// ---- POUs/LVCP2/PRG_LVCP2_CompensationCalculate.TcPOU
PROGRAM PRG_LVCP2_CompensationCalculate
VAR
    fbCompensationCalc : FB_CompensationCalculator;
    bCalculate : BOOL := TRUE;              // Sürekli hesaplama için
    nActiveGroups : INT := 10;              // Toplam 10 grup
    
    // Outputs
    stHMIData : ST_CompensationHMI;
    asCapacitorTags : ARRAY[0..99] OF STRING(30);
    nActiveTags : INT;
    
    // Özet bilgiler
    rTotalPower : REAL;
    nTotalCapacitors : INT;
    nActiveGroupCount : INT;
END_VAR

// Grup sayısını güncelle
GVL_LVCP1.nConfiguredGroups := nActiveGroups;

// Hesaplama
fbCompensationCalc(
    bExecute 				:= bCalculate,
    bGroupActive 			:= GVL_LVCP2.abGroupActive,
    stGroupConfig 			:= GVL_LVCP2.astCompensationGroups,
    nActiveGroups 			:= GVL_LVCP2.nConfiguredGroups,
    stHMI 					=> stHMIData,
    asActiveCapacitorTags 	=> asCapacitorTags,
    nActiveCapacitorCount 	=> nActiveTags
);

// Özet bilgiler
rTotalPower 		:= stHMIData.stSummary.rTotalActivePower;
nTotalCapacitors 	:= stHMIData.stSummary.nTotalActiveCapacitors;
nActiveGroupCount 	:= stHMIData.stSummary.nActiveGroupCount;

END_PROGRAM

// ---- POUs/LVCP2/PRG_LVCP2_MainDisconnector.TcPOU
PROGRAM PRG_LVCP2_MainDisconnector
VAR
    // Function Block Instance
    fbDisconnector		: FB_DisconnectorControl;
	
	stDisconnectorIO	: ST_DisconnectorIO;
	
    
    // Başlangıç konfigürasyonu için flag
    bInitDone: BOOL := FALSE;	
END_VAR

IF NOT bInitDone THEN
	bInitDone := TRUE;
	RETURN;
END_IF

//*************************************************************************
// Ana Besleme Ayırıcısı
// +EP7-8CB1
//*************************************************************************
fbDisconnector(
    // Fiziksel Girişler
    bContactorOn_FB 	:= stDisconnectorIO.bContactorOn_FB,
    bContactorOff_FB 	:= stDisconnectorIO.bContactorOff_FB,
    bLimitOn 			:= stDisconnectorIO.bLimitOn,
    bLimitOff 			:= stDisconnectorIO.bLimitOff,
    bThermalFault 		:= stDisconnectorIO.bThermalFault,
    bEarthSwitchOn 		:= stDisconnectorIO.bEarthSwitchOn,
    bEarthSwitchOff 	:= stDisconnectorIO.bEarthSwitchOff,
    bPLCControl 		:= stDisconnectorIO.bPLCControl,
    
    // Güvenlik Girişleri
    bSafetyLoop 		:= GVL_Alarm.bSafetyLoop,
    bInterlock 			:= FALSE,
    
    // Sistem Girişleri
    bMasterReset 		:= GVL_Alarm.bMasterReset,
    
    // HMI Bağlantısı
    stHMI 				:= GVL_LVCP2.stMainDisconnectorHMI,
    
    // Fiziksel Çıkışlar
    bContactorOn_Out 	=> stDisconnectorIO.bContactorOn_Out,
    bContactorOff_Out 	=> stDisconnectorIO.bContactorOff_Out
);

METHOD M_Init : BOOL
VAR_INPUT
END_VAR

GVL_LVCP1.stMainDisconnectorHMI.stConfig.bEarthSwitchExists := TRUE;
GVL_LVCP1.stMainDisconnectorHMI.stConfig.bGrounded := TRUE;
GVL_LVCP1.stMainDisconnectorHMI.stConfig.bInterlockEnable := TRUE;
GVL_LVCP1.stMainDisconnectorHMI.stConfig.dwOperationLimit := 10000;
GVL_LVCP1.stMainDisconnectorHMI.stConfig.nPhaseCount := 3;
GVL_LVCP1.stMainDisconnectorHMI.stConfig.rRatedCurrent := 1600.0;
GVL_LVCP1.stMainDisconnectorHMI.stConfig.rRatedVoltage := 1000.0;
GVL_LVCP1.stMainDisconnectorHMI.stConfig.sProductCode := '';
GVL_LVCP1.stMainDisconnectorHMI.stConfig.sProjectCode := '+EP7-8CB1';
GVL_LVCP1.stMainDisconnectorHMI.stConfig.tContactorDelay := T#500MS;
GVL_LVCP1.stMainDisconnectorHMI.stConfig.tMotionTimeout := T#50S;
END_METHOD

END_PROGRAM

// ---- POUs/LVCP2/PRG_LVCP2_Colors.TcPOU
PROGRAM PRG_LVCP2_Colors
VAR
	arrLine : ARRAY[1..4] OF E_LineColors;
	arrCapacitorSchemaColor : ARRAY[1..10] OF ST_CapacitorSchemaColorWithContactor;

	i : INT;
	bInitDone : BOOL;
END_VAR

IF NOT bInitDone THEN
	ACT_ContactorConfigurations();
	bInitDone := TRUE;
END_IF

//line1
arrLine[1] := E_LineColors.Energised_Red;

//line2
arrLine[2] := arrLine[1];

//line3
arrLine[3] := arrLine[2];

//line4
arrLine[4] := arrLine[3];

//şemaları kendi içerisinde kontrol edicez
FOR i:=1 TO 10 DO
	arrCapacitorSchemaColor[i].GroundColor := E_LineColors.Grounded_Green;
	arrCapacitorSchemaColor[i].BottomLineColor2 := E_LineColors.Grounded_Green;

	//topline
	arrCapacitorSchemaColor[i].TopLineColor := arrLine[4];
	
	//bottomLine - şema üzerinde ayırıcının altındaki her iki line birbiri ile bağlantılı olduğu için tek yerden yönetiliyor
	IF arrCapacitorSchemaColor[i].ContactorPosition = E_ContactorPosition.ON THEN
		arrCapacitorSchemaColor[i].BottomLineColor := arrCapacitorSchemaColor[i].TopLineColor;
	ELSE
		arrCapacitorSchemaColor[i].BottomLineColor := E_LineColors.Default;
	END_IF
	
	//capacitor
	arrCapacitorSchemaColor[i].CapacitorColor := arrCapacitorSchemaColor[i].BottomLineColor;
	
END_FOR

ACTION ACT_ContactorConfigurations:
arrCapacitorSchemaColor[1].ContactorPosition := GVL_LVCP2.stGroup1_ContactorHMI.stStatus.ePosition;
arrCapacitorSchemaColor[2].ContactorPosition := GVL_LVCP2.stGroup2_ContactorHMI.stStatus.ePosition;
arrCapacitorSchemaColor[3].ContactorPosition := GVL_LVCP2.stGroup3_ContactorHMI.stStatus.ePosition;
arrCapacitorSchemaColor[4].ContactorPosition := GVL_LVCP2.stGroup4_ContactorHMI.stStatus.ePosition;
arrCapacitorSchemaColor[5].ContactorPosition := GVL_LVCP2.stGroup5_ContactorHMI.stStatus.ePosition;
arrCapacitorSchemaColor[6].ContactorPosition := GVL_LVCP2.stGroup6_ContactorHMI.stStatus.ePosition;
arrCapacitorSchemaColor[7].ContactorPosition := GVL_LVCP2.stGroup7_ContactorHMI.stStatus.ePosition;
arrCapacitorSchemaColor[8].ContactorPosition := GVL_LVCP2.stGroup8_ContactorHMI.stStatus.ePosition;
arrCapacitorSchemaColor[9].ContactorPosition := GVL_LVCP2.stGroup9_ContactorHMI.stStatus.ePosition;
arrCapacitorSchemaColor[10].ContactorPosition := GVL_LVCP2.stGroup10_ContactorHMI.stStatus.ePosition;
END_ACTION

END_PROGRAM

// ---- POUs/LVCP2/PRG_LVCP2_Group1.TcPOU
PROGRAM PRG_LVCP2_Group1
VAR
    // Function Block Instance
    fbContactor: FB_ContactorControl;

    // Contactor 1 IO Structure  
    stContactor_IO: ST_ContactorIO;
    
    // Başlangıç konfigürasyonu için flag
    bContactorInitDone: BOOL := FALSE;
    bCapacitorInitDone: BOOL := FALSE;	
END_VAR



	M_Contactor();
	
	M_Capacitor();

METHOD M_Capacitor : BOOL
VAR
    nGroupIndex : INT;
END_VAR
	nGroupIndex := 0;  // Grup 1 için index
	
	IF NOT bCapacitorInitDone THEN
	
		// Grup 1 değerlerini ata
		GVL_LVCP2.astCompensationGroups[nGroupIndex].rPower := 25.0;
		GVL_LVCP2.astCompensationGroups[nGroupIndex].rVoltage := 450.0;
		GVL_LVCP2.astCompensationGroups[nGroupIndex].nQuantity := 10;
		GVL_LVCP2.astCompensationGroups[nGroupIndex].sTagPrefix := '+EP7-16C1';
		GVL_LVCP2.astCompensationGroups[nGroupIndex].sProductCode := 'ENT.CXD-450-25';
		
		bCapacitorInitDone := TRUE;
	END_IF
	
	// Grup 1 aktif durumu
	GVL_LVCP2.abGroupActive[nGroupIndex] := stContactor_IO.bFeedback;
	
	M_Capacitor := TRUE;
END_METHOD

METHOD M_Contactor : BOOL
VAR_INPUT
END_VAR
IF NOT bContactorInitDone THEN
    // Konfigürasyon parametreleri
    GVL_LVCP2.stGroup1_ContactorHMI.stConfig.sProjectCode := '+EP7-17K1';
    GVL_LVCP2.stGroup1_ContactorHMI.stConfig.sProductCode := 'ABB-1SFL637001R7011';
    GVL_LVCP2.stGroup1_ContactorHMI.stConfig.rRatedCurrent := 630.0;
    GVL_LVCP2.stGroup1_ContactorHMI.stConfig.rRatedVoltage := 1000.0;
    GVL_LVCP2.stGroup1_ContactorHMI.stConfig.nPhaseCount := 3;
    GVL_LVCP2.stGroup1_ContactorHMI.stConfig.tFeedbackDelay := T#500MS;
    GVL_LVCP2.stGroup1_ContactorHMI.stConfig.tWeldedDelay := T#2S;
    GVL_LVCP2.stGroup1_ContactorHMI.stConfig.dwOperationLimit := 100000;
    GVL_LVCP2.stGroup1_ContactorHMI.stConfig.bFeedbackRequired := FALSE;
    // Başlangıç bakım sayacı
    GVL_LVCP2.stGroup1_ContactorHMI.stStatistics.dwRemainingOperations := GVL_LVCP2.stGroup1_ContactorHMI.stConfig.dwOperationLimit;
	
	bContactorInitDone := TRUE;
END_IF	
	
// Function Block Çağrısı
fbContactor(
    // Fiziksel Girişler
    bFeedback 		:= stContactor_IO.bFeedback,
    bPLCControl 	:= stContactor_IO.bPLCControl,
    
    // Güvenlik Girişleri
    bSafetyLoop 	:= GVL_Alarm.bSafetyLoop,
    bInterlock 		:= FALSE,
    
    // Sistem Girişleri
    bMasterReset 	:= GVL_Alarm.bMasterReset,
    
    // HMI Bağlantısı
    stHMI 			:= GVL_LVCP2.stGroup1_ContactorHMI,
    
    // Fiziksel Çıkış
    bOutput 		=> stContactor_IO.bOutput
);

// SQL Kayıt İşlemi
IF GVL_LVCP2.stGroup1_ContactorHMI.stStatistics.bNewOperationFlag THEN
    // SQL kayıt fonksiyonunu çağır
    GVL_LVCP2.stGroup1_ContactorHMI.stStatistics.bNewOperationFlag := FALSE;
END_IF
END_METHOD

END_PROGRAM

// ---- POUs/LVCP2/PRG_LVCP2_Group2.TcPOU
PROGRAM PRG_LVCP2_Group2
VAR
    // Function Block Instance
    fbContactor: FB_ContactorControl;

    // Contactor 1 IO Structure  
    stContactor_IO: ST_ContactorIO;
    
    // Başlangıç konfigürasyonu için flag
    bContactorInitDone: BOOL := FALSE;
    bCapacitorInitDone: BOOL := FALSE;	
END_VAR



	M_Contactor();
	
	M_Capacitor();

METHOD M_Capacitor : BOOL
VAR
    nGroupIndex : INT;
END_VAR

nGroupIndex := 1;  // Grup 2 için index

IF NOT bCapacitorInitDone THEN
    // Grup 2 değerlerini ata
    GVL_LVCP2.astCompensationGroups[nGroupIndex].rPower := 25.0;
    GVL_LVCP2.astCompensationGroups[nGroupIndex].rVoltage := 450.0;
    GVL_LVCP2.astCompensationGroups[nGroupIndex].nQuantity := 8;
    GVL_LVCP2.astCompensationGroups[nGroupIndex].sTagPrefix := '+EP7-19C1';
    GVL_LVCP2.astCompensationGroups[nGroupIndex].sProductCode := 'ENT.CXD-450-25';
    
    bCapacitorInitDone := TRUE;
END_IF

// Grup 2 aktif durumu
GVL_LVCP2.abGroupActive[nGroupIndex] := stContactor_IO.bFeedback;

M_Capacitor := TRUE;
END_METHOD

METHOD M_Contactor : BOOL
VAR_INPUT
END_VAR

IF NOT bContactorInitDone THEN
    // Konfigürasyon parametreleri
    GVL_LVCP2.stGroup2_ContactorHMI.stConfig.sProjectCode := '+EP7-20K1';
    GVL_LVCP2.stGroup2_ContactorHMI.stConfig.sProductCode := 'ABB-1SFL597001R7011';
    GVL_LVCP2.stGroup2_ContactorHMI.stConfig.rRatedCurrent := 500.0;
    GVL_LVCP2.stGroup2_ContactorHMI.stConfig.rRatedVoltage := 1000.0;
    GVL_LVCP2.stGroup2_ContactorHMI.stConfig.nPhaseCount := 3;
    GVL_LVCP2.stGroup2_ContactorHMI.stConfig.tFeedbackDelay := T#500MS;
    GVL_LVCP2.stGroup2_ContactorHMI.stConfig.tWeldedDelay := T#2S;
    GVL_LVCP2.stGroup2_ContactorHMI.stConfig.dwOperationLimit := 100000;
    
    // Başlangıç bakım sayacı
    GVL_LVCP2.stGroup2_ContactorHMI.stStatistics.dwRemainingOperations := GVL_LVCP2.stGroup2_ContactorHMI.stConfig.dwOperationLimit;
    
    bContactorInitDone := TRUE;
END_IF

// Function Block Çağrısı
fbContactor(
    // Fiziksel Girişler
    bFeedback := stContactor_IO.bFeedback,
    bPLCControl := stContactor_IO.bPLCControl,
    
    // Güvenlik Girişleri
    bSafetyLoop := GVL_Alarm.bSafetyLoop,
    bInterlock := FALSE,
    
    // Sistem Girişleri
    bMasterReset := GVL_Alarm.bMasterReset,
    
    // HMI Bağlantısı
    stHMI := GVL_LVCP2.stGroup2_ContactorHMI,
    
    // Fiziksel Çıkış
    bOutput => stContactor_IO.bOutput
);

M_Contactor := TRUE;
END_METHOD

END_PROGRAM

// ---- POUs/LVCP2/PRG_LVCP2_Group3.TcPOU
PROGRAM PRG_LVCP2_Group3
VAR
    // Function Block Instance
    fbContactor: FB_ContactorControl;

    // Contactor 1 IO Structure  
    stContactor_IO: ST_ContactorIO;
    
    // Başlangıç konfigürasyonu için flag
    bContactorInitDone: BOOL := FALSE;
    bCapacitorInitDone: BOOL := FALSE;	
END_VAR



	M_Contactor();
	
	M_Capacitor();

METHOD M_Capacitor : BOOL
VAR
    nGroupIndex : INT;
END_VAR

nGroupIndex := 2;  // Grup 3 için index

IF NOT bCapacitorInitDone THEN
    // Grup 3 değerlerini ata
    GVL_LVCP2.astCompensationGroups[nGroupIndex].rPower := 25.0;
    GVL_LVCP2.astCompensationGroups[nGroupIndex].rVoltage := 450.0;
    GVL_LVCP2.astCompensationGroups[nGroupIndex].nQuantity := 6;
    GVL_LVCP2.astCompensationGroups[nGroupIndex].sTagPrefix := '+EP7-22C1';
    GVL_LVCP2.astCompensationGroups[nGroupIndex].sProductCode := 'ENT.CXD-450-25';
    
    bCapacitorInitDone := TRUE;
END_IF

// Grup 3 aktif durumu
GVL_LVCP2.abGroupActive[nGroupIndex] := stContactor_IO.bFeedback;

M_Capacitor := TRUE;
END_METHOD

METHOD M_Contactor : BOOL
VAR_INPUT
END_VAR
IF NOT bContactorInitDone THEN
    // Konfigürasyon parametreleri
    GVL_LVCP2.stGroup3_ContactorHMI.stConfig.sProjectCode := '+EP7-23K1';
    GVL_LVCP2.stGroup3_ContactorHMI.stConfig.sProductCode := 'ABB-1SFL597001R7011';
    GVL_LVCP2.stGroup3_ContactorHMI.stConfig.rRatedCurrent := 500.0;
    GVL_LVCP2.stGroup3_ContactorHMI.stConfig.rRatedVoltage := 1000.0;
    GVL_LVCP2.stGroup3_ContactorHMI.stConfig.nPhaseCount := 3;
    GVL_LVCP2.stGroup3_ContactorHMI.stConfig.tFeedbackDelay := T#500MS;
    GVL_LVCP2.stGroup3_ContactorHMI.stConfig.tWeldedDelay := T#2S;
    GVL_LVCP2.stGroup3_ContactorHMI.stConfig.dwOperationLimit := 100000;
    
    // Başlangıç bakım sayacı
    GVL_LVCP2.stGroup3_ContactorHMI.stStatistics.dwRemainingOperations := GVL_LVCP2.stGroup3_ContactorHMI.stConfig.dwOperationLimit;
    
    bContactorInitDone := TRUE;
END_IF

// Function Block Çağrısı
fbContactor(
    // Fiziksel Girişler
    bFeedback := stContactor_IO.bFeedback,
    bPLCControl := stContactor_IO.bPLCControl,
    
    // Güvenlik Girişleri
    bSafetyLoop := GVL_Alarm.bSafetyLoop,
    bInterlock := FALSE,
    
    // Sistem Girişleri
    bMasterReset := GVL_Alarm.bMasterReset,
    
    // HMI Bağlantısı
    stHMI := GVL_LVCP2.stGroup3_ContactorHMI,
    
    // Fiziksel Çıkış
    bOutput => stContactor_IO.bOutput
);

M_Contactor := TRUE;
END_METHOD

END_PROGRAM

// ---- POUs/LVCP2/PRG_LVCP2_Group4.TcPOU
PROGRAM PRG_LVCP2_Group4
VAR
    // Function Block Instance
    fbContactor: FB_ContactorControl;

    // Contactor 1 IO Structure  
    stContactor_IO: ST_ContactorIO;
    
    // Başlangıç konfigürasyonu için flag
    bContactorInitDone: BOOL := FALSE;
    bCapacitorInitDone: BOOL := FALSE;	
END_VAR



	M_Contactor();
	
	M_Capacitor();

METHOD M_Capacitor : BOOL
VAR
    nGroupIndex : INT;
END_VAR

nGroupIndex := 3;  // Grup 4 için index

IF NOT bCapacitorInitDone THEN
    // Grup 4 değerlerini ata
    GVL_LVCP2.astCompensationGroups[nGroupIndex].rPower := 25.0;
    GVL_LVCP2.astCompensationGroups[nGroupIndex].rVoltage := 450.0;
    GVL_LVCP2.astCompensationGroups[nGroupIndex].nQuantity := 5;
    GVL_LVCP2.astCompensationGroups[nGroupIndex].sTagPrefix := '+EP7-25C1';
    GVL_LVCP2.astCompensationGroups[nGroupIndex].sProductCode := 'ENT.CXD-450-25';
    
    bCapacitorInitDone := TRUE;
END_IF

// Grup 4 aktif durumu
GVL_LVCP2.abGroupActive[nGroupIndex] := stContactor_IO.bFeedback;

M_Capacitor := TRUE;
END_METHOD

METHOD M_Contactor : BOOL
VAR_INPUT
END_VAR
IF NOT bContactorInitDone THEN
    // Konfigürasyon parametreleri
    GVL_LVCP2.stGroup4_ContactorHMI.stConfig.sProjectCode := '+EP7-26K1';
    GVL_LVCP2.stGroup4_ContactorHMI.stConfig.sProductCode := 'ABB-1SFL597001R7011';
    GVL_LVCP2.stGroup4_ContactorHMI.stConfig.rRatedCurrent := 500.0;
    GVL_LVCP2.stGroup4_ContactorHMI.stConfig.rRatedVoltage := 1000.0;
    GVL_LVCP2.stGroup4_ContactorHMI.stConfig.nPhaseCount := 3;
    GVL_LVCP2.stGroup4_ContactorHMI.stConfig.tFeedbackDelay := T#500MS;
    GVL_LVCP2.stGroup4_ContactorHMI.stConfig.tWeldedDelay := T#2S;
    GVL_LVCP2.stGroup4_ContactorHMI.stConfig.dwOperationLimit := 100000;
    
    // Başlangıç bakım sayacı
    GVL_LVCP2.stGroup4_ContactorHMI.stStatistics.dwRemainingOperations := GVL_LVCP2.stGroup4_ContactorHMI.stConfig.dwOperationLimit;
    
    bContactorInitDone := TRUE;
END_IF

// Function Block Çağrısı
fbContactor(
    // Fiziksel Girişler
    bFeedback := stContactor_IO.bFeedback,
    bPLCControl := stContactor_IO.bPLCControl,
    
    // Güvenlik Girişleri
    bSafetyLoop := GVL_Alarm.bSafetyLoop,
    bInterlock := FALSE,
    
    // Sistem Girişleri
    bMasterReset := GVL_Alarm.bMasterReset,
    
    // HMI Bağlantısı
    stHMI := GVL_LVCP2.stGroup4_ContactorHMI,
    
    // Fiziksel Çıkış
    bOutput => stContactor_IO.bOutput
);

M_Contactor := TRUE;
END_METHOD

END_PROGRAM

// ---- POUs/LVCP2/PRG_LVCP2_Group5.TcPOU
PROGRAM PRG_LVCP2_Group5
VAR
    // Function Block Instance
    fbContactor: FB_ContactorControl;

    // Contactor 1 IO Structure  
    stContactor_IO: ST_ContactorIO;
    
    // Başlangıç konfigürasyonu için flag
    bContactorInitDone: BOOL := FALSE;
    bCapacitorInitDone: BOOL := FALSE;	
END_VAR



	M_Contactor();
	
	M_Capacitor();

METHOD M_Capacitor : BOOL
VAR
    nGroupIndex : INT;
END_VAR

nGroupIndex := 4;  // Grup 5 için index

IF NOT bCapacitorInitDone THEN
    // Grup 5 değerlerini ata
    GVL_LVCP2.astCompensationGroups[nGroupIndex].rPower := 25.0;
    GVL_LVCP2.astCompensationGroups[nGroupIndex].rVoltage := 450.0;
    GVL_LVCP2.astCompensationGroups[nGroupIndex].nQuantity := 4;
    GVL_LVCP2.astCompensationGroups[nGroupIndex].sTagPrefix := '+EP7-28C1';
    GVL_LVCP2.astCompensationGroups[nGroupIndex].sProductCode := 'ENT.CXD-450-25';
    
    bCapacitorInitDone := TRUE;
END_IF

// Grup 5 aktif durumu
GVL_LVCP2.abGroupActive[nGroupIndex] := stContactor_IO.bFeedback;

M_Capacitor := TRUE;
END_METHOD

METHOD M_Contactor : BOOL
VAR_INPUT
END_VAR
IF NOT bContactorInitDone THEN
    // Konfigürasyon parametreleri
    GVL_LVCP2.stGroup5_ContactorHMI.stConfig.sProjectCode := '+EP7-29K1';
    GVL_LVCP2.stGroup5_ContactorHMI.stConfig.sProductCode := 'ABB 1SFL547002R1311';
    GVL_LVCP2.stGroup5_ContactorHMI.stConfig.rRatedCurrent := 265.0;
    GVL_LVCP2.stGroup5_ContactorHMI.stConfig.rRatedVoltage := 1000.0;
    GVL_LVCP2.stGroup5_ContactorHMI.stConfig.nPhaseCount := 3;
    GVL_LVCP2.stGroup5_ContactorHMI.stConfig.tFeedbackDelay := T#500MS;
    GVL_LVCP2.stGroup5_ContactorHMI.stConfig.tWeldedDelay := T#2S;
    GVL_LVCP2.stGroup5_ContactorHMI.stConfig.dwOperationLimit := 100000;
    
    // Başlangıç bakım sayacı
    GVL_LVCP2.stGroup5_ContactorHMI.stStatistics.dwRemainingOperations := GVL_LVCP2.stGroup5_ContactorHMI.stConfig.dwOperationLimit;
    
    bContactorInitDone := TRUE;
END_IF

// Function Block Çağrısı
fbContactor(
    // Fiziksel Girişler
    bFeedback := stContactor_IO.bFeedback,
    bPLCControl := stContactor_IO.bPLCControl,
    
    // Güvenlik Girişleri
    bSafetyLoop := GVL_Alarm.bSafetyLoop,
    bInterlock := FALSE,
    
    // Sistem Girişleri
    bMasterReset := GVL_Alarm.bMasterReset,
    
    // HMI Bağlantısı
    stHMI := GVL_LVCP2.stGroup5_ContactorHMI,
    
    // Fiziksel Çıkış
    bOutput => stContactor_IO.bOutput
);

M_Contactor := TRUE;
END_METHOD

END_PROGRAM

// ---- POUs/LVCP2/PRG_LVCP2_Group6.TcPOU
PROGRAM PRG_LVCP2_Group6
VAR
    // Function Block Instance
    fbContactor: FB_ContactorControl;

    // Contactor 1 IO Structure  
    stContactor_IO: ST_ContactorIO;
    
    // Başlangıç konfigürasyonu için flag
    bContactorInitDone: BOOL := FALSE;
    bCapacitorInitDone: BOOL := FALSE;	
END_VAR



	M_Contactor();
	
	M_Capacitor();

METHOD M_Capacitor : BOOL
VAR
    nGroupIndex : INT;
END_VAR

nGroupIndex := 5;  // Grup 6 için index

IF NOT bCapacitorInitDone THEN
    // Grup 6 değerlerini ata
    GVL_LVCP2.astCompensationGroups[nGroupIndex].rPower := 25.0;
    GVL_LVCP2.astCompensationGroups[nGroupIndex].rVoltage := 450.0;
    GVL_LVCP2.astCompensationGroups[nGroupIndex].nQuantity := 3;
    GVL_LVCP2.astCompensationGroups[nGroupIndex].sTagPrefix := '+EP7-31C1';
    GVL_LVCP2.astCompensationGroups[nGroupIndex].sProductCode := 'ENT.CXD-450-25';
    
    bCapacitorInitDone := TRUE;
END_IF

// Grup 6 aktif durumu
GVL_LVCP2.abGroupActive[nGroupIndex] := stContactor_IO.bFeedback;

M_Capacitor := TRUE;
END_METHOD

METHOD M_Contactor : BOOL
VAR_INPUT
END_VAR
IF NOT bContactorInitDone THEN
    // Konfigürasyon parametreleri
    GVL_LVCP2.stGroup6_ContactorHMI.stConfig.sProjectCode := '+EP7-30K1';
    GVL_LVCP2.stGroup6_ContactorHMI.stConfig.sProductCode := 'ABB 1SFL547002R1311';
    GVL_LVCP2.stGroup6_ContactorHMI.stConfig.rRatedCurrent := 265.0;
    GVL_LVCP2.stGroup6_ContactorHMI.stConfig.rRatedVoltage := 1000.0;
    GVL_LVCP2.stGroup6_ContactorHMI.stConfig.nPhaseCount := 3;
    GVL_LVCP2.stGroup6_ContactorHMI.stConfig.tFeedbackDelay := T#500MS;
    GVL_LVCP2.stGroup6_ContactorHMI.stConfig.tWeldedDelay := T#2S;
    GVL_LVCP2.stGroup6_ContactorHMI.stConfig.dwOperationLimit := 100000;
    
    // Başlangıç bakım sayacı
    GVL_LVCP2.stGroup6_ContactorHMI.stStatistics.dwRemainingOperations := GVL_LVCP2.stGroup6_ContactorHMI.stConfig.dwOperationLimit;
    
    bContactorInitDone := TRUE;
END_IF

// Function Block Çağrısı
fbContactor(
    // Fiziksel Girişler
    bFeedback := stContactor_IO.bFeedback,
    bPLCControl := stContactor_IO.bPLCControl,
    
    // Güvenlik Girişleri
    bSafetyLoop := GVL_Alarm.bSafetyLoop,
    bInterlock := FALSE,
    
    // Sistem Girişleri
    bMasterReset := GVL_Alarm.bMasterReset,
    
    // HMI Bağlantısı
    stHMI := GVL_LVCP2.stGroup6_ContactorHMI,
    
    // Fiziksel Çıkış
    bOutput => stContactor_IO.bOutput
);

M_Contactor := TRUE;
END_METHOD

END_PROGRAM

// ---- POUs/LVCP2/PRG_LVCP2_Group7.TcPOU
PROGRAM PRG_LVCP2_Group7
VAR
    // Function Block Instance
    fbContactor: FB_ContactorControl;

    // Contactor 1 IO Structure  
    stContactor_IO: ST_ContactorIO;
    
    // Başlangıç konfigürasyonu için flag
    bContactorInitDone: BOOL := FALSE;
    bCapacitorInitDone: BOOL := FALSE;	
END_VAR



	M_Contactor();
	
	M_Capacitor();

METHOD M_Capacitor : BOOL
VAR
    nGroupIndex : INT;
END_VAR

nGroupIndex := 6;  // Grup 7 için index

IF NOT bCapacitorInitDone THEN
    // Grup 7 değerlerini ata
    GVL_LVCP2.astCompensationGroups[nGroupIndex].rPower := 25.0;
    GVL_LVCP2.astCompensationGroups[nGroupIndex].rVoltage := 450.0;
    GVL_LVCP2.astCompensationGroups[nGroupIndex].nQuantity := 2;
    GVL_LVCP2.astCompensationGroups[nGroupIndex].sTagPrefix := '+EP7-34C1';
    GVL_LVCP2.astCompensationGroups[nGroupIndex].sProductCode := 'ENT.CXD-450-25';
    
    bCapacitorInitDone := TRUE;
END_IF

// Grup 7 aktif durumu
GVL_LVCP2.abGroupActive[nGroupIndex] := stContactor_IO.bFeedback;

M_Capacitor := TRUE;
END_METHOD

METHOD M_Contactor : BOOL
VAR_INPUT
END_VAR
IF NOT bContactorInitDone THEN
    // Konfigürasyon parametreleri
    GVL_LVCP2.stGroup7_ContactorHMI.stConfig.sProjectCode := '+EP7-35K1';
    GVL_LVCP2.stGroup7_ContactorHMI.stConfig.sProductCode := 'ABB 1SFL447001R1311';
    GVL_LVCP2.stGroup7_ContactorHMI.stConfig.rRatedCurrent := 150.0;
    GVL_LVCP2.stGroup7_ContactorHMI.stConfig.rRatedVoltage := 1000.0;
    GVL_LVCP2.stGroup7_ContactorHMI.stConfig.nPhaseCount := 3;
    GVL_LVCP2.stGroup7_ContactorHMI.stConfig.tFeedbackDelay := T#500MS;
    GVL_LVCP2.stGroup7_ContactorHMI.stConfig.tWeldedDelay := T#2S;
    GVL_LVCP2.stGroup7_ContactorHMI.stConfig.dwOperationLimit := 100000;
    
    // Başlangıç bakım sayacı
    GVL_LVCP2.stGroup7_ContactorHMI.stStatistics.dwRemainingOperations := GVL_LVCP2.stGroup7_ContactorHMI.stConfig.dwOperationLimit;
    
    bContactorInitDone := TRUE;
END_IF

// Function Block Çağrısı
fbContactor(
    // Fiziksel Girişler
    bFeedback := stContactor_IO.bFeedback,
    bPLCControl := stContactor_IO.bPLCControl,
    
    // Güvenlik Girişleri
    bSafetyLoop := GVL_Alarm.bSafetyLoop,
    bInterlock := FALSE,
    
    // Sistem Girişleri
    bMasterReset := GVL_Alarm.bMasterReset,
    
    // HMI Bağlantısı
    stHMI := GVL_LVCP2.stGroup7_ContactorHMI,
    
    // Fiziksel Çıkış
    bOutput => stContactor_IO.bOutput
);

M_Contactor := TRUE;
END_METHOD

END_PROGRAM

// ---- POUs/LVCP2/PRG_LVCP2_Group8.TcPOU
PROGRAM PRG_LVCP2_Group8
VAR
    // Function Block Instance
    fbContactor: FB_ContactorControl;

    // Contactor 1 IO Structure  
    stContactor_IO: ST_ContactorIO;
    
    // Başlangıç konfigürasyonu için flag
    bContactorInitDone: BOOL := FALSE;
    bCapacitorInitDone: BOOL := FALSE;	
END_VAR



	M_Contactor();
	
	M_Capacitor();

METHOD M_Capacitor : BOOL
VAR
    nGroupIndex : INT;
END_VAR

nGroupIndex := 7;  // Grup 8 için index

IF NOT bCapacitorInitDone THEN
    // Grup 8 değerlerini ata
    GVL_LVCP2.astCompensationGroups[nGroupIndex].rPower := 12.5;
    GVL_LVCP2.astCompensationGroups[nGroupIndex].rVoltage := 450.0;
    GVL_LVCP2.astCompensationGroups[nGroupIndex].nQuantity := 3;
    GVL_LVCP2.astCompensationGroups[nGroupIndex].sTagPrefix := '+EP7-37C1';
    GVL_LVCP2.astCompensationGroups[nGroupIndex].sProductCode := 'ENT.CXD-450-12.5';
    
    bCapacitorInitDone := TRUE;
END_IF

// Grup 8 aktif durumu
GVL_LVCP2.abGroupActive[nGroupIndex] := stContactor_IO.bFeedback;

M_Capacitor := TRUE;
END_METHOD

METHOD M_Contactor : BOOL
VAR_INPUT
END_VAR
IF NOT bContactorInitDone THEN
    // Konfigürasyon parametreleri
    GVL_LVCP2.stGroup8_ContactorHMI.stConfig.sProjectCode := '+EP7-38K1';
    GVL_LVCP2.stGroup8_ContactorHMI.stConfig.sProductCode := 'ABB 1SFL447001R1311';
    GVL_LVCP2.stGroup8_ContactorHMI.stConfig.rRatedCurrent := 115.0;
    GVL_LVCP2.stGroup8_ContactorHMI.stConfig.rRatedVoltage := 1000.0;
    GVL_LVCP2.stGroup8_ContactorHMI.stConfig.nPhaseCount := 3;
    GVL_LVCP2.stGroup8_ContactorHMI.stConfig.tFeedbackDelay := T#500MS;
    GVL_LVCP2.stGroup8_ContactorHMI.stConfig.tWeldedDelay := T#2S;
    GVL_LVCP2.stGroup8_ContactorHMI.stConfig.dwOperationLimit := 100000;
    
    // Başlangıç bakım sayacı
    GVL_LVCP2.stGroup8_ContactorHMI.stStatistics.dwRemainingOperations := GVL_LVCP2.stGroup8_ContactorHMI.stConfig.dwOperationLimit;
    
    bContactorInitDone := TRUE;
END_IF

// Function Block Çağrısı
fbContactor(
    // Fiziksel Girişler
    bFeedback := stContactor_IO.bFeedback,
    bPLCControl := stContactor_IO.bPLCControl,
    
    // Güvenlik Girişleri
    bSafetyLoop := GVL_Alarm.bSafetyLoop,
    bInterlock := FALSE,
    
    // Sistem Girişleri
    bMasterReset := GVL_Alarm.bMasterReset,
    
    // HMI Bağlantısı
    stHMI := GVL_LVCP2.stGroup8_ContactorHMI,
    
    // Fiziksel Çıkış
    bOutput => stContactor_IO.bOutput
);

M_Contactor := TRUE;
END_METHOD

END_PROGRAM

// ---- POUs/LVCP2/PRG_LVCP2_Group9.TcPOU
PROGRAM PRG_LVCP2_Group9
VAR
    // Function Block Instance
    fbContactor: FB_ContactorControl;

    // Contactor 1 IO Structure  
    stContactor_IO: ST_ContactorIO;
    
    // Başlangıç konfigürasyonu için flag
    bContactorInitDone: BOOL := FALSE;
    bCapacitorInitDone: BOOL := FALSE;	
END_VAR



	M_Contactor();
	
	M_Capacitor();

METHOD M_Capacitor : BOOL
VAR
    nGroupIndex : INT;
END_VAR

nGroupIndex := 8;  // Grup 9 için index

IF NOT bCapacitorInitDone THEN
    // Grup 9 değerlerini ata
    GVL_LVCP2.astCompensationGroups[nGroupIndex].rPower := 12.5;
    GVL_LVCP2.astCompensationGroups[nGroupIndex].rVoltage := 450.0;
    GVL_LVCP2.astCompensationGroups[nGroupIndex].nQuantity := 2;
    GVL_LVCP2.astCompensationGroups[nGroupIndex].sTagPrefix := '+EP7-40C1';
    GVL_LVCP2.astCompensationGroups[nGroupIndex].sProductCode := 'ENT.CXD-450-12.5';
    
    bCapacitorInitDone := TRUE;
END_IF

// Grup 9 aktif durumu
GVL_LVCP2.abGroupActive[nGroupIndex] := stContactor_IO.bFeedback;

M_Capacitor := TRUE;
END_METHOD

METHOD M_Contactor : BOOL
VAR_INPUT
END_VAR
IF NOT bContactorInitDone THEN
    // Konfigürasyon parametreleri
    GVL_LVCP2.stGroup9_ContactorHMI.stConfig.sProjectCode := '+EP7-41K1';
    GVL_LVCP2.stGroup9_ContactorHMI.stConfig.sProductCode := 'ABB 1SFL427001R1311';
    GVL_LVCP2.stGroup9_ContactorHMI.stConfig.rRatedCurrent := 115.0;
    GVL_LVCP2.stGroup9_ContactorHMI.stConfig.rRatedVoltage := 1000.0;
    GVL_LVCP2.stGroup9_ContactorHMI.stConfig.nPhaseCount := 3;
    GVL_LVCP2.stGroup9_ContactorHMI.stConfig.tFeedbackDelay := T#500MS;
    GVL_LVCP2.stGroup9_ContactorHMI.stConfig.tWeldedDelay := T#2S;
    GVL_LVCP2.stGroup9_ContactorHMI.stConfig.dwOperationLimit := 100000;
    
    // Başlangıç bakım sayacı
    GVL_LVCP2.stGroup9_ContactorHMI.stStatistics.dwRemainingOperations := GVL_LVCP2.stGroup9_ContactorHMI.stConfig.dwOperationLimit;
    
    bContactorInitDone := TRUE;
END_IF

// Function Block Çağrısı
fbContactor(
    // Fiziksel Girişler
    bFeedback := stContactor_IO.bFeedback,
    bPLCControl := stContactor_IO.bPLCControl,
    
    // Güvenlik Girişleri
    bSafetyLoop := GVL_Alarm.bSafetyLoop,
    bInterlock := FALSE,
    
    // Sistem Girişleri
    bMasterReset := GVL_Alarm.bMasterReset,
    
    // HMI Bağlantısı
    stHMI := GVL_LVCP2.stGroup9_ContactorHMI,
    
    // Fiziksel Çıkış
    bOutput => stContactor_IO.bOutput
);

M_Contactor := TRUE;
END_METHOD

END_PROGRAM

// ---- POUs/LVCP2/PRG_LVCP2_Group10.TcPOU
PROGRAM PRG_LVCP2_Group10
VAR
    // Function Block Instance
    fbContactor: FB_ContactorControl;

    // Contactor 1 IO Structure  
    stContactor_IO: ST_ContactorIO;
    
    // Başlangıç konfigürasyonu için flag
    bContactorInitDone: BOOL := FALSE;
    bCapacitorInitDone: BOOL := FALSE;	
END_VAR



	M_Contactor();
	
	M_Capacitor();

METHOD M_Capacitor : BOOL
VAR
    nGroupIndex : INT;
END_VAR

nGroupIndex := 9;  // Grup 10 için index

IF NOT bCapacitorInitDone THEN
    // Grup 10 değerlerini ata
    GVL_LVCP2.astCompensationGroups[nGroupIndex].rPower := 12.5;
    GVL_LVCP2.astCompensationGroups[nGroupIndex].rVoltage := 450.0;
    GVL_LVCP2.astCompensationGroups[nGroupIndex].nQuantity := 1;
    GVL_LVCP2.astCompensationGroups[nGroupIndex].sTagPrefix := '+EP7-43C1';
    GVL_LVCP2.astCompensationGroups[nGroupIndex].sProductCode := 'ENT.CXD-450-12.5';
    
    bCapacitorInitDone := TRUE;
END_IF

// Grup 10 aktif durumu
GVL_LVCP2.abGroupActive[nGroupIndex] := stContactor_IO.bFeedback;

M_Capacitor := TRUE;
END_METHOD

METHOD M_Contactor : BOOL
VAR_INPUT
END_VAR
IF NOT bContactorInitDone THEN
    // Konfigürasyon parametreleri
    GVL_LVCP2.stGroup10_ContactorHMI.stConfig.sProjectCode := '+EP7-43K1';
    GVL_LVCP2.stGroup10_ContactorHMI.stConfig.sProductCode := 'ABB 1SFL427001R1311';
    GVL_LVCP2.stGroup10_ContactorHMI.stConfig.rRatedCurrent := 115.0;
    GVL_LVCP2.stGroup10_ContactorHMI.stConfig.rRatedVoltage := 1000.0;
    GVL_LVCP2.stGroup10_ContactorHMI.stConfig.nPhaseCount := 3;
    GVL_LVCP2.stGroup10_ContactorHMI.stConfig.tFeedbackDelay := T#500MS;
    GVL_LVCP2.stGroup10_ContactorHMI.stConfig.tWeldedDelay := T#2S;
    GVL_LVCP2.stGroup10_ContactorHMI.stConfig.dwOperationLimit := 100000;
    
    // Başlangıç bakım sayacı
    GVL_LVCP2.stGroup10_ContactorHMI.stStatistics.dwRemainingOperations := GVL_LVCP2.stGroup10_ContactorHMI.stConfig.dwOperationLimit;
    
    bContactorInitDone := TRUE;
END_IF

// Function Block Çağrısı
fbContactor(
    // Fiziksel Girişler
    bFeedback := stContactor_IO.bFeedback,
    bPLCControl := stContactor_IO.bPLCControl,
    
    // Güvenlik Girişleri
    bSafetyLoop := GVL_Alarm.bSafetyLoop,
    bInterlock := FALSE,
    
    // Sistem Girişleri
    bMasterReset := GVL_Alarm.bMasterReset,
    
    // HMI Bağlantısı
    stHMI := GVL_LVCP2.stGroup10_ContactorHMI,
    
    // Fiziksel Çıkış
    bOutput => stContactor_IO.bOutput
);

M_Contactor := TRUE;
END_METHOD

END_PROGRAM

// ---- POUs/LVCP5/PRG_LVCP5.TcPOU
PROGRAM PRG_LVCP5
VAR
END_VAR

	PRG_LVCP5_PowerMeasurement();

 	PRG_LVCP5_CompensationCalculate();

	PRG_LVCP5_MainCircuitBreaker();
	
	PRG_LVCP5_Colors();
	
	PRG_LVCP5_Group1();
	
	PRG_LVCP5_Group2();
	
	PRG_LVCP5_Group3();	
	
	PRG_LVCP5_Group4();	

	PRG_LVCP5_Group5();	

	PRG_LVCP5_Group6();	

	PRG_LVCP5_Group7();

END_PROGRAM

// ---- POUs/LVCP5/PRG_LVCP5_PowerMeasurement.TcPOU
PROGRAM PRG_LVCP5_PowerMeasurement
VAR
	// Enerji Yönetimi
	fbEL3453	: FB_EL3453;	
	stEL3453	: stEL3453;
END_VAR


	fbEL3453(pOut := ADR(stEL3453));

END_PROGRAM

// ---- POUs/LVCP5/PRG_LVCP5_CompensationCalculate.TcPOU
PROGRAM PRG_LVCP5_CompensationCalculate
VAR
    fbCompensationCalc : FB_CompensationCalculator;
    bCalculate : BOOL := TRUE;              // Sürekli hesaplama için
    nActiveGroups : INT := 10;              // Toplam 10 grup
    
    // Outputs
    stHMIData : ST_CompensationHMI;
    asCapacitorTags : ARRAY[0..99] OF STRING(30);
    nActiveTags : INT;
    
    // Özet bilgiler
    rTotalPower : REAL;
    nTotalCapacitors : INT;
    nActiveGroupCount : INT;
END_VAR

// Grup sayısını güncelle
GVL_LVCP5.nConfiguredGroups := nActiveGroups;

// Hesaplama
fbCompensationCalc(
    bExecute 				:= bCalculate,
    bGroupActive 			:= GVL_LVCP5.abGroupActive,
    stGroupConfig 			:= GVL_LVCP5.astCompensationGroups,
    nActiveGroups 			:= GVL_LVCP5.nConfiguredGroups,
    stHMI 					=> stHMIData,
    asActiveCapacitorTags 	=> asCapacitorTags,
    nActiveCapacitorCount 	=> nActiveTags
);

// Özet bilgiler
rTotalPower 		:= stHMIData.stSummary.rTotalActivePower;
nTotalCapacitors 	:= stHMIData.stSummary.nTotalActiveCapacitors;
nActiveGroupCount 	:= stHMIData.stSummary.nActiveGroupCount;

END_PROGRAM

// ---- POUs/LVCP5/PRG_LVCP5_MainCircuitBreaker.TcPOU
PROGRAM PRG_LVCP5_MainCircuitBreaker
VAR
    // Function Block Instance
    fbCircuitBreaker	: FB_CircuitBreaker;
	
    // IO Structure
    stCircuitBreakerIO	: ST_CircuitBreakerIO;	
    
    // Başlangıç konfigürasyonu için flag
    bInitDone			: BOOL := FALSE;
END_VAR

IF NOT bInitDone THEN
	M_Init();
	bInitDone := TRUE;
END_IF

// Function Block Çağrısı
fbCircuitBreaker(
    // Fiziksel Girişler
    bPositionOn 		:= stCircuitBreakerIO.bPositionOn,
    bPositionOff 		:= stCircuitBreakerIO.bPositionOff,
    bPositionTripped 	:= stCircuitBreakerIO.bPositionTripped,
    bSpringCharged 		:= stCircuitBreakerIO.bSpringCharged,
    bPLCControl 		:= stCircuitBreakerIO.bPLCControl,
    
    // Güvenlik Girişleri
    bSafetyLoop 		:= GVL_Alarm.bSafetyLoop,
    bInterlock 			:= FALSE,
    
    // Sistem Girişleri
    bMasterReset 		:= GVL_Alarm.bMasterReset,
    
    // HMI Bağlantısı
    stHMI 				:= GVL_LVCP5.stMainCircuitBreakerHMI,
    
    // Fiziksel Çıkışlar
    bOnCommand 			=> stCircuitBreakerIO.bOnCommand,
    bOffCommand 		=> stCircuitBreakerIO.bOffCommand
);

// SQL Kayıt İşlemi
IF GVL_LVCP5.stMainCircuitBreakerHMI.stStatistics.bNewOperationFlag THEN
    // SQL kayıt fonksiyonunu çağır
    GVL_LVCP5.stMainCircuitBreakerHMI.stStatistics.bNewOperationFlag := FALSE;
END_IF

METHOD M_Init : BOOL
VAR_INPUT
END_VAR
    // Konfigürasyon parametreleri
    GVL_LVCP5.stMainCircuitBreakerHMI.stConfig.sProjectCode := '+EP8-6F1';
    GVL_LVCP5.stMainCircuitBreakerHMI.stConfig.sProductCode := 'ETN C63N32D630';
    GVL_LVCP5.stMainCircuitBreakerHMI.stConfig.rRatedCurrent := 630.0;
    GVL_LVCP5.stMainCircuitBreakerHMI.stConfig.rRatedVoltage := 1000.0;
    GVL_LVCP5.stMainCircuitBreakerHMI.stConfig.nPhaseCount := 3;
    GVL_LVCP5.stMainCircuitBreakerHMI.stConfig.tMotionTimeout := T#5S;
    GVL_LVCP5.stMainCircuitBreakerHMI.stConfig.tSpringChargeTimeout := T#30S;
    GVL_LVCP5.stMainCircuitBreakerHMI.stConfig.bSpringChargeRequired := FALSE;
    GVL_LVCP5.stMainCircuitBreakerHMI.stConfig.dwOperationLimit := 10000;
    
    // Başlangıç bakım sayacı
    GVL_LVCP5.stMainCircuitBreakerHMI.stStatistics.dwRemainingOperations := GVL_LVCP5.stMainCircuitBreakerHMI.stConfig.dwOperationLimit;
END_METHOD

END_PROGRAM

// ---- POUs/LVCP5/PRG_LVCP5_Colors.TcPOU
PROGRAM PRG_LVCP5_Colors
VAR
	arrLine : ARRAY[1..4] OF E_LineColors;
	arrCapacitorSchemaColor : ARRAY[1..7] OF ST_CapacitorSchemaColorWithContactor;

	i : INT;
	bInitDone : BOOL;
END_VAR

IF NOT bInitDone THEN
	ACT_ContactorConfigurations();
	bInitDone := TRUE;
END_IF

//line1
arrLine[1] := E_LineColors.Energised_Red;

//line2
arrLine[2] := arrLine[1];

//line3
arrLine[3] := arrLine[2];

//line4
arrLine[4] := arrLine[3];

//şemaları kendi içerisinde kontrol edicez
FOR i:=1 TO 10 DO
	arrCapacitorSchemaColor[i].GroundColor := E_LineColors.Grounded_Green;
	arrCapacitorSchemaColor[i].BottomLineColor2 := E_LineColors.Grounded_Green;

	//topline
	arrCapacitorSchemaColor[i].TopLineColor := arrLine[4];
	
	//bottomLine - şema üzerinde ayırıcının altındaki her iki line birbiri ile bağlantılı olduğu için tek yerden yönetiliyor
	IF arrCapacitorSchemaColor[i].ContactorPosition = E_ContactorPosition.ON THEN
		arrCapacitorSchemaColor[i].BottomLineColor := arrCapacitorSchemaColor[i].TopLineColor;
	ELSE
		arrCapacitorSchemaColor[i].BottomLineColor := E_LineColors.Default;
	END_IF
	
	//capacitor
	arrCapacitorSchemaColor[i].CapacitorColor := arrCapacitorSchemaColor[i].BottomLineColor;
	
END_FOR

ACTION ACT_ContactorConfigurations:
arrCapacitorSchemaColor[1].ContactorPosition := GVL_LVCP5.stGroup1_ContactorHMI.stStatus.ePosition;
arrCapacitorSchemaColor[2].ContactorPosition := GVL_LVCP5.stGroup2_ContactorHMI.stStatus.ePosition;
arrCapacitorSchemaColor[3].ContactorPosition := GVL_LVCP5.stGroup3_ContactorHMI.stStatus.ePosition;
arrCapacitorSchemaColor[4].ContactorPosition := GVL_LVCP5.stGroup4_ContactorHMI.stStatus.ePosition;
arrCapacitorSchemaColor[5].ContactorPosition := GVL_LVCP5.stGroup5_ContactorHMI.stStatus.ePosition;
arrCapacitorSchemaColor[6].ContactorPosition := GVL_LVCP5.stGroup6_ContactorHMI.stStatus.ePosition;
arrCapacitorSchemaColor[7].ContactorPosition := GVL_LVCP5.stGroup7_ContactorHMI.stStatus.ePosition;
END_ACTION

END_PROGRAM

// ---- POUs/LVCP5/PRG_LVCP5_Group1.TcPOU
PROGRAM PRG_LVCP5_Group1
VAR
    // Function Block Instance
    fbContactor: FB_ContactorControl;

    // Contactor 1 IO Structure  
    stContactor_IO: ST_ContactorIO;
    
    // Başlangıç konfigürasyonu için flag
    bContactorInitDone: BOOL := FALSE;
    bCapacitorInitDone: BOOL := FALSE;	
END_VAR



	M_Contactor();
	
	M_Capacitor();

METHOD M_Capacitor : BOOL
VAR
    nGroupIndex : INT;
END_VAR
	nGroupIndex := 0;  // Grup 1 için index
	
	IF NOT bCapacitorInitDone THEN
	
		// Grup 1 değerlerini ata
		GVL_LVCP5.astCompensationGroups[nGroupIndex].rPower := 10.0;
		GVL_LVCP5.astCompensationGroups[nGroupIndex].rVoltage := 450.0;
		GVL_LVCP5.astCompensationGroups[nGroupIndex].nQuantity := 10;
		GVL_LVCP5.astCompensationGroups[nGroupIndex].sTagPrefix := '+EP8-16C1';
		GVL_LVCP5.astCompensationGroups[nGroupIndex].sProductCode := 'ENT.CXD-450-10';
		
		bCapacitorInitDone := TRUE;
	END_IF
	
	// Grup 1 aktif durumu
	GVL_LVCP5.abGroupActive[nGroupIndex] := stContactor_IO.bFeedback;
	
	M_Capacitor := TRUE;
END_METHOD

METHOD M_Contactor : BOOL
VAR_INPUT
END_VAR
IF NOT bContactorInitDone THEN
    // Konfigürasyon parametreleri
    GVL_LVCP5.stGroup1_ContactorHMI.stConfig.sProjectCode := '+EP8-17K1';
    GVL_LVCP5.stGroup1_ContactorHMI.stConfig.sProductCode := 'SCH LC1G225LSEA';
    GVL_LVCP5.stGroup1_ContactorHMI.stConfig.rRatedCurrent := 225.0;
    GVL_LVCP5.stGroup1_ContactorHMI.stConfig.rRatedVoltage := 1000.0;
    GVL_LVCP5.stGroup1_ContactorHMI.stConfig.nPhaseCount := 3;
    GVL_LVCP5.stGroup1_ContactorHMI.stConfig.tFeedbackDelay := T#500MS;
    GVL_LVCP5.stGroup1_ContactorHMI.stConfig.tWeldedDelay := T#2S;
    GVL_LVCP5.stGroup1_ContactorHMI.stConfig.dwOperationLimit := 100000;
    
    // Başlangıç bakım sayacı
    GVL_LVCP5.stGroup1_ContactorHMI.stStatistics.dwRemainingOperations := GVL_LVCP5.stGroup1_ContactorHMI.stConfig.dwOperationLimit;
	
	bContactorInitDone := TRUE;
END_IF	
	
// Function Block Çağrısı
fbContactor(
    // Fiziksel Girişler
    bFeedback 		:= stContactor_IO.bFeedback,
    bPLCControl 	:= stContactor_IO.bPLCControl,
    
    // Güvenlik Girişleri
    bSafetyLoop 	:= GVL_Alarm.bSafetyLoop,
    bInterlock 		:= FALSE,
    
    // Sistem Girişleri
    bMasterReset 	:= GVL_Alarm.bMasterReset,
    
    // HMI Bağlantısı
    stHMI 			:= GVL_LVCP5.stGroup1_ContactorHMI,
    
    // Fiziksel Çıkış
    bOutput 		=> stContactor_IO.bOutput
);

// SQL Kayıt İşlemi
IF GVL_LVCP5.stGroup1_ContactorHMI.stStatistics.bNewOperationFlag THEN
    // SQL kayıt fonksiyonunu çağır
    GVL_LVCP5.stGroup1_ContactorHMI.stStatistics.bNewOperationFlag := FALSE;
END_IF
END_METHOD

END_PROGRAM

// ---- POUs/LVCP5/PRG_LVCP5_Group2.TcPOU
PROGRAM PRG_LVCP5_Group2
VAR
    // Function Block Instance
    fbContactor: FB_ContactorControl;

    // Contactor 1 IO Structure  
    stContactor_IO: ST_ContactorIO;
    
    // Başlangıç konfigürasyonu için flag
    bContactorInitDone: BOOL := FALSE;
    bCapacitorInitDone: BOOL := FALSE;	
END_VAR



	M_Contactor();
	
	M_Capacitor();

METHOD M_Capacitor : BOOL
VAR
    nGroupIndex : INT;
END_VAR

nGroupIndex := 1;  // Grup 2 için index

IF NOT bCapacitorInitDone THEN
    // Grup 2 değerlerini ata
    GVL_LVCP5.astCompensationGroups[nGroupIndex].rPower := 10.0;
    GVL_LVCP5.astCompensationGroups[nGroupIndex].rVoltage := 450.0;
    GVL_LVCP5.astCompensationGroups[nGroupIndex].nQuantity := 9;
    GVL_LVCP5.astCompensationGroups[nGroupIndex].sTagPrefix := '+EP8-19C1';
    GVL_LVCP5.astCompensationGroups[nGroupIndex].sProductCode := 'ENT.CXD-450-10';
    
    bCapacitorInitDone := TRUE;
END_IF

// Grup 2 aktif durumu
GVL_LVCP5.abGroupActive[nGroupIndex] := stContactor_IO.bFeedback;

M_Capacitor := TRUE;
END_METHOD

METHOD M_Contactor : BOOL
VAR_INPUT
END_VAR

IF NOT bContactorInitDone THEN
    // Konfigürasyon parametreleri
    GVL_LVCP5.stGroup2_ContactorHMI.stConfig.sProjectCode := '+EP6-20K1';
    GVL_LVCP5.stGroup2_ContactorHMI.stConfig.sProductCode := 'SCH LC1G500LSEA';
    GVL_LVCP5.stGroup2_ContactorHMI.stConfig.rRatedCurrent := 500.0;
    GVL_LVCP5.stGroup2_ContactorHMI.stConfig.rRatedVoltage := 1000.0;
    GVL_LVCP5.stGroup2_ContactorHMI.stConfig.nPhaseCount := 3;
    GVL_LVCP5.stGroup2_ContactorHMI.stConfig.tFeedbackDelay := T#500MS;
    GVL_LVCP5.stGroup2_ContactorHMI.stConfig.tWeldedDelay := T#2S;
    GVL_LVCP5.stGroup2_ContactorHMI.stConfig.dwOperationLimit := 100000;
    
    // Başlangıç bakım sayacı
    GVL_LVCP5.stGroup2_ContactorHMI.stStatistics.dwRemainingOperations := GVL_LVCP5.stGroup2_ContactorHMI.stConfig.dwOperationLimit;
    
    bContactorInitDone := TRUE;
END_IF

// Function Block Çağrısı
fbContactor(
    // Fiziksel Girişler
    bFeedback 		:= stContactor_IO.bFeedback,
    bPLCControl 	:= stContactor_IO.bPLCControl,
    
    // Güvenlik Girişleri
    bSafetyLoop 	:= GVL_Alarm.bSafetyLoop,
    bInterlock 		:= FALSE,
    
    // Sistem Girişleri
    bMasterReset 	:= GVL_Alarm.bMasterReset,
    
    // HMI Bağlantısı
    stHMI 			:= GVL_LVCP5.stGroup2_ContactorHMI,
    
    // Fiziksel Çıkış
    bOutput 		=> stContactor_IO.bOutput
);

M_Contactor := TRUE;
END_METHOD

END_PROGRAM

// ---- POUs/LVCP5/PRG_LVCP5_Group3.TcPOU
PROGRAM PRG_LVCP5_Group3
VAR
    // Function Block Instance
    fbContactor: FB_ContactorControl;

    // Contactor 1 IO Structure  
    stContactor_IO: ST_ContactorIO;
    
    // Başlangıç konfigürasyonu için flag
    bContactorInitDone: BOOL := FALSE;
    bCapacitorInitDone: BOOL := FALSE;	
END_VAR



	M_Contactor();
	
	M_Capacitor();

METHOD M_Capacitor : BOOL
VAR
    nGroupIndex : INT;
END_VAR

nGroupIndex := 2;  // Grup 3 için index

IF NOT bCapacitorInitDone THEN
    // Grup 3 değerlerini ata
    GVL_LVCP5.astCompensationGroups[nGroupIndex].rPower := 10.0;
    GVL_LVCP5.astCompensationGroups[nGroupIndex].rVoltage := 450.0;
    GVL_LVCP5.astCompensationGroups[nGroupIndex].nQuantity := 8;
    GVL_LVCP5.astCompensationGroups[nGroupIndex].sTagPrefix := '+EP8-22C1';
    GVL_LVCP5.astCompensationGroups[nGroupIndex].sProductCode := 'ENT.CXD-450-10';
    
    bCapacitorInitDone := TRUE;
END_IF

// Grup 3 aktif durumu
GVL_LVCP5.abGroupActive[nGroupIndex] := stContactor_IO.bFeedback;

M_Capacitor := TRUE;
END_METHOD

METHOD M_Contactor : BOOL
VAR_INPUT
END_VAR
IF NOT bContactorInitDone THEN
    // Konfigürasyon parametreleri
    GVL_LVCP5.stGroup3_ContactorHMI.stConfig.sProjectCode := '+EP8-23K1';
    GVL_LVCP5.stGroup3_ContactorHMI.stConfig.sProductCode := 'SCH LC1G185LSEA';
    GVL_LVCP5.stGroup3_ContactorHMI.stConfig.rRatedCurrent := 185.0;
    GVL_LVCP5.stGroup3_ContactorHMI.stConfig.rRatedVoltage := 1000.0;
    GVL_LVCP5.stGroup3_ContactorHMI.stConfig.nPhaseCount := 3;
    GVL_LVCP5.stGroup3_ContactorHMI.stConfig.tFeedbackDelay := T#500MS;
    GVL_LVCP5.stGroup3_ContactorHMI.stConfig.tWeldedDelay := T#2S;
    GVL_LVCP5.stGroup3_ContactorHMI.stConfig.dwOperationLimit := 100000;
    
    // Başlangıç bakım sayacı
    GVL_LVCP5.stGroup3_ContactorHMI.stStatistics.dwRemainingOperations := GVL_LVCP5.stGroup3_ContactorHMI.stConfig.dwOperationLimit;
    
    bContactorInitDone := TRUE;
END_IF

// Function Block Çağrısı
fbContactor(
    // Fiziksel Girişler
    bFeedback 		:= stContactor_IO.bFeedback,
    bPLCControl 	:= stContactor_IO.bPLCControl,
    
    // Güvenlik Girişleri
    bSafetyLoop 	:= GVL_Alarm.bSafetyLoop,
    bInterlock 		:= FALSE,
    
    // Sistem Girişleri
    bMasterReset 	:= GVL_Alarm.bMasterReset,
    
    // HMI Bağlantısı
    stHMI 			:= GVL_LVCP5.stGroup3_ContactorHMI,
    
    // Fiziksel Çıkış
    bOutput 		=> stContactor_IO.bOutput
);

M_Contactor := TRUE;
END_METHOD

END_PROGRAM

// ---- POUs/LVCP5/PRG_LVCP5_Group4.TcPOU
PROGRAM PRG_LVCP5_Group4
VAR
    // Function Block Instance
    fbContactor: FB_ContactorControl;

    // Contactor 1 IO Structure  
    stContactor_IO: ST_ContactorIO;
    
    // Başlangıç konfigürasyonu için flag
    bContactorInitDone: BOOL := FALSE;
    bCapacitorInitDone: BOOL := FALSE;	
END_VAR



	M_Contactor();
	
	M_Capacitor();

METHOD M_Capacitor : BOOL
VAR
    nGroupIndex : INT;
END_VAR

nGroupIndex := 3;  // Grup 4 için index

IF NOT bCapacitorInitDone THEN
    // Grup 4 değerlerini ata
    GVL_LVCP5.astCompensationGroups[nGroupIndex].rPower := 10.0;
    GVL_LVCP5.astCompensationGroups[nGroupIndex].rVoltage := 450.0;
    GVL_LVCP5.astCompensationGroups[nGroupIndex].nQuantity := 7;
    GVL_LVCP5.astCompensationGroups[nGroupIndex].sTagPrefix := '+EP8-25C1';
    GVL_LVCP5.astCompensationGroups[nGroupIndex].sProductCode := 'ENT.CXD-450-10';
    
    bCapacitorInitDone := TRUE;
END_IF

// Grup 4 aktif durumu
GVL_LVCP5.abGroupActive[nGroupIndex] := stContactor_IO.bFeedback;

M_Capacitor := TRUE;
END_METHOD

METHOD M_Contactor : BOOL
VAR_INPUT
END_VAR
IF NOT bContactorInitDone THEN
    // Konfigürasyon parametreleri
    GVL_LVCP5.stGroup4_ContactorHMI.stConfig.sProjectCode := '+EP8-26K1';
    GVL_LVCP5.stGroup4_ContactorHMI.stConfig.sProductCode := 'SCH LC1G150LSEA';
    GVL_LVCP5.stGroup4_ContactorHMI.stConfig.rRatedCurrent := 150.0;
    GVL_LVCP5.stGroup4_ContactorHMI.stConfig.rRatedVoltage := 1000.0;
    GVL_LVCP5.stGroup4_ContactorHMI.stConfig.nPhaseCount := 3;
    GVL_LVCP5.stGroup4_ContactorHMI.stConfig.tFeedbackDelay := T#500MS;
    GVL_LVCP5.stGroup4_ContactorHMI.stConfig.tWeldedDelay := T#2S;
    GVL_LVCP5.stGroup4_ContactorHMI.stConfig.dwOperationLimit := 100000;
    
    // Başlangıç bakım sayacı
    GVL_LVCP5.stGroup4_ContactorHMI.stStatistics.dwRemainingOperations := GVL_LVCP5.stGroup4_ContactorHMI.stConfig.dwOperationLimit;
    
    bContactorInitDone := TRUE;
END_IF

// Function Block Çağrısı
fbContactor(
    // Fiziksel Girişler
    bFeedback 		:= stContactor_IO.bFeedback,
    bPLCControl 	:= stContactor_IO.bPLCControl,
    
    // Güvenlik Girişleri
    bSafetyLoop 	:= GVL_Alarm.bSafetyLoop,
    bInterlock 		:= FALSE,
    
    // Sistem Girişleri
    bMasterReset 	:= GVL_Alarm.bMasterReset,
    
    // HMI Bağlantısı
    stHMI 			:= GVL_LVCP5.stGroup4_ContactorHMI,
    
    // Fiziksel Çıkış
    bOutput 		=> stContactor_IO.bOutput
);

M_Contactor := TRUE;
END_METHOD

END_PROGRAM

// ---- POUs/LVCP5/PRG_LVCP5_Group5.TcPOU
PROGRAM PRG_LVCP5_Group5
VAR
    // Function Block Instance
    fbContactor: FB_ContactorControl;

    // Contactor 1 IO Structure  
    stContactor_IO: ST_ContactorIO;
    
    // Başlangıç konfigürasyonu için flag
    bContactorInitDone: BOOL := FALSE;
    bCapacitorInitDone: BOOL := FALSE;	
END_VAR

	M_Contactor();
	
	M_Capacitor();

METHOD M_Capacitor : BOOL
VAR
    nGroupIndex : INT;
END_VAR

nGroupIndex := 4;  // Grup 5 için index

IF NOT bCapacitorInitDone THEN
    // Grup 5 değerlerini ata
    GVL_LVCP5.astCompensationGroups[nGroupIndex].rPower := 10.0;
    GVL_LVCP5.astCompensationGroups[nGroupIndex].rVoltage := 450.0;
    GVL_LVCP5.astCompensationGroups[nGroupIndex].nQuantity := 3;
    GVL_LVCP5.astCompensationGroups[nGroupIndex].sTagPrefix := '+EP8-28C1';
    GVL_LVCP5.astCompensationGroups[nGroupIndex].sProductCode := 'ENT.CXD-450-10';
    
    bCapacitorInitDone := TRUE;
END_IF

// Grup 5 aktif durumu
GVL_LVCP5.abGroupActive[nGroupIndex] := stContactor_IO.bFeedback;

M_Capacitor := TRUE;
END_METHOD

METHOD M_Contactor : BOOL
VAR_INPUT
END_VAR
bContactorInitDone := bContactorInitDone;
IF NOT bContactorInitDone THEN
    // Konfigürasyon parametreleri
    GVL_LVCP5.stGroup5_ContactorHMI.stConfig.sProjectCode := '+EP8-29K1';
    GVL_LVCP5.stGroup5_ContactorHMI.stConfig.sProductCode := 'SCH LC1D40A3P7';
    GVL_LVCP5.stGroup5_ContactorHMI.stConfig.rRatedCurrent := 40.0;
    GVL_LVCP5.stGroup5_ContactorHMI.stConfig.rRatedVoltage := 690.0;
    GVL_LVCP5.stGroup5_ContactorHMI.stConfig.nPhaseCount := 3;
    GVL_LVCP5.stGroup5_ContactorHMI.stConfig.tFeedbackDelay := T#500MS;
    GVL_LVCP5.stGroup5_ContactorHMI.stConfig.tWeldedDelay := T#2S;
    GVL_LVCP5.stGroup5_ContactorHMI.stConfig.dwOperationLimit := 100000;
    
    // Başlangıç bakım sayacı
    GVL_LVCP5.stGroup5_ContactorHMI.stStatistics.dwRemainingOperations := GVL_LVCP5.stGroup5_ContactorHMI.stConfig.dwOperationLimit;
    
    bContactorInitDone := TRUE;
END_IF

// Function Block Çağrısı
fbContactor(
    // Fiziksel Girişler
    bFeedback 		:= stContactor_IO.bFeedback,
    bPLCControl 	:= stContactor_IO.bPLCControl,
    
    // Güvenlik Girişleri
    bSafetyLoop 	:= GVL_Alarm.bSafetyLoop,
    bInterlock 		:= FALSE,
    
    // Sistem Girişleri
    bMasterReset 	:= GVL_Alarm.bMasterReset,
    
    // HMI Bağlantısı
    stHMI 			:= GVL_LVCP5.stGroup5_ContactorHMI,
    
    // Fiziksel Çıkış
    bOutput 		=> stContactor_IO.bOutput
);

M_Contactor := TRUE;
END_METHOD

END_PROGRAM

// ---- POUs/LVCP5/PRG_LVCP5_Group6.TcPOU
PROGRAM PRG_LVCP5_Group6
VAR
    // Function Block Instance
    fbContactor: FB_ContactorControl;

    // Contactor 1 IO Structure  
    stContactor_IO: ST_ContactorIO;
    
    // Başlangıç konfigürasyonu için flag
    bContactorInitDone: BOOL := FALSE;
    bCapacitorInitDone: BOOL := FALSE;	
END_VAR



	M_Contactor();
	
	M_Capacitor();

METHOD M_Capacitor : BOOL
VAR
    nGroupIndex : INT;
END_VAR

nGroupIndex := 5;  // Grup 6 için index

IF NOT bCapacitorInitDone THEN
    // Grup 6 değerlerini ata
    GVL_LVCP5.astCompensationGroups[nGroupIndex].rPower := 25.0;
    GVL_LVCP5.astCompensationGroups[nGroupIndex].rVoltage := 450.0;
    GVL_LVCP5.astCompensationGroups[nGroupIndex].nQuantity := 2;
    GVL_LVCP5.astCompensationGroups[nGroupIndex].sTagPrefix := '+EP8-31C1';
    GVL_LVCP5.astCompensationGroups[nGroupIndex].sProductCode := 'ENT.CXD-450-10';
    
    bCapacitorInitDone := TRUE;
END_IF

// Grup 6 aktif durumu
GVL_LVCP5.abGroupActive[nGroupIndex] := stContactor_IO.bFeedback;

M_Capacitor := TRUE;
END_METHOD

METHOD M_Contactor : BOOL
VAR_INPUT
END_VAR
IF NOT bContactorInitDone THEN
    // Konfigürasyon parametreleri
    GVL_LVCP5.stGroup6_ContactorHMI.stConfig.sProjectCode := '+EP8-32K1';
    GVL_LVCP5.stGroup6_ContactorHMI.stConfig.sProductCode := 'SCH LC1D40A3P7';
    GVL_LVCP5.stGroup6_ContactorHMI.stConfig.rRatedCurrent := 40.0;
    GVL_LVCP5.stGroup6_ContactorHMI.stConfig.rRatedVoltage := 690.0;
    GVL_LVCP5.stGroup6_ContactorHMI.stConfig.nPhaseCount := 3;
    GVL_LVCP5.stGroup6_ContactorHMI.stConfig.tFeedbackDelay := T#500MS;
    GVL_LVCP5.stGroup6_ContactorHMI.stConfig.tWeldedDelay := T#2S;
    GVL_LVCP5.stGroup6_ContactorHMI.stConfig.dwOperationLimit := 100000;
    
    // Başlangıç bakım sayacı
    GVL_LVCP5.stGroup6_ContactorHMI.stStatistics.dwRemainingOperations := GVL_LVCP5.stGroup6_ContactorHMI.stConfig.dwOperationLimit;
    
    bContactorInitDone := TRUE;
END_IF

// Function Block Çağrısı
fbContactor(
    // Fiziksel Girişler
    bFeedback 		:= stContactor_IO.bFeedback,
    bPLCControl 	:= stContactor_IO.bPLCControl,
    
    // Güvenlik Girişleri
    bSafetyLoop 	:= GVL_Alarm.bSafetyLoop,
    bInterlock 		:= FALSE,
    
    // Sistem Girişleri
    bMasterReset 	:= GVL_Alarm.bMasterReset,
    
    // HMI Bağlantısı
    stHMI 			:= GVL_LVCP5.stGroup6_ContactorHMI,
    
    // Fiziksel Çıkış
    bOutput 		=> stContactor_IO.bOutput
);

M_Contactor := TRUE;
END_METHOD

END_PROGRAM

// ---- POUs/LVCP5/PRG_LVCP5_Group7.TcPOU
PROGRAM PRG_LVCP5_Group7
VAR
    // Function Block Instance
    fbContactor: FB_ContactorControl;

    // Contactor 1 IO Structure  
    stContactor_IO: ST_ContactorIO;
    
    // Başlangıç konfigürasyonu için flag
    bContactorInitDone: BOOL := FALSE;
    bCapacitorInitDone: BOOL := FALSE;	
END_VAR



	M_Contactor();
	
	M_Capacitor();

METHOD M_Capacitor : BOOL
VAR
    nGroupIndex : INT;
END_VAR

nGroupIndex := 6;  // Grup 7 için index

IF NOT bCapacitorInitDone THEN
    // Grup 7 değerlerini ata
    GVL_LVCP5.astCompensationGroups[nGroupIndex].rPower := 10.0;
    GVL_LVCP5.astCompensationGroups[nGroupIndex].rVoltage := 450.0;
    GVL_LVCP5.astCompensationGroups[nGroupIndex].nQuantity := 1;
    GVL_LVCP5.astCompensationGroups[nGroupIndex].sTagPrefix := '+EP8-34C1';
    GVL_LVCP5.astCompensationGroups[nGroupIndex].sProductCode := 'ENT.CXD-450-10';
    
    bCapacitorInitDone := TRUE;
END_IF

// Grup 7 aktif durumu
GVL_LVCP5.abGroupActive[nGroupIndex] := stContactor_IO.bFeedback;

M_Capacitor := TRUE;
END_METHOD

METHOD M_Contactor : BOOL
VAR_INPUT
END_VAR
IF NOT bContactorInitDone THEN
    // Konfigürasyon parametreleri
    GVL_LVCP5.stGroup7_ContactorHMI.stConfig.sProjectCode := '+EP6-35K1';
    GVL_LVCP5.stGroup7_ContactorHMI.stConfig.sProductCode := 'SCH LC1D25P7';
    GVL_LVCP5.stGroup7_ContactorHMI.stConfig.rRatedCurrent := 25.0;
    GVL_LVCP5.stGroup7_ContactorHMI.stConfig.rRatedVoltage := 690.0;
    GVL_LVCP5.stGroup7_ContactorHMI.stConfig.nPhaseCount := 3;
    GVL_LVCP5.stGroup7_ContactorHMI.stConfig.tFeedbackDelay := T#500MS;
    GVL_LVCP5.stGroup7_ContactorHMI.stConfig.tWeldedDelay := T#2S;
    GVL_LVCP5.stGroup7_ContactorHMI.stConfig.dwOperationLimit := 100000;
    
    // Başlangıç bakım sayacı
    GVL_LVCP5.stGroup7_ContactorHMI.stStatistics.dwRemainingOperations := GVL_LVCP5.stGroup7_ContactorHMI.stConfig.dwOperationLimit;
    
    bContactorInitDone := TRUE;
END_IF

// Function Block Çağrısı
fbContactor(
    // Fiziksel Girişler
    bFeedback 		:= stContactor_IO.bFeedback,
    bPLCControl 	:= stContactor_IO.bPLCControl,
    
    // Güvenlik Girişleri
    bSafetyLoop 	:= GVL_Alarm.bSafetyLoop,
    bInterlock 		:= FALSE,
    
    // Sistem Girişleri
    bMasterReset 	:= GVL_Alarm.bMasterReset,
    
    // HMI Bağlantısı
    stHMI 			:= GVL_LVCP5.stGroup7_ContactorHMI,
    
    // Fiziksel Çıkış
    bOutput 		=> stContactor_IO.bOutput
);

M_Contactor := TRUE;
END_METHOD

END_PROGRAM

// ---- POUs/HVCP3/PRG_HVCP3.TcPOU
PROGRAM PRG_HVCP3
VAR
END_VAR

	PRG_HVCP3_10CB1();
	
PRG_HVCP3_12CB1();

PRG_HVCP3_14CB1();	

PRG_HVCP3_16CB1();

PRG_HVCP3_18CB1();

PRG_HVCP3_20CB1();

PRG_HVCP3_22CB1();

PRG_HVCP3_24CB1();

PRG_HVCP3_26CB1();

PRG_HVCP3_28CB1();

PRG_HVCP3_30CB1();

PRG_HVCP3_32CB1();

PRG_HVCP3_34CB1();

PRG_HVCP3_36CB1();

PRG_HVCP3_38CB1();

PRG_HVCP3_40CB1();

PRG_HVCP3_42CB1();

PRG_HVCP3_44CB1();

PRG_HVCP3_46CB1();

PRG_HVCP3_48CB1();

PRG_HVCP3_50CB1();

PRG_HVCP3_52CB1();

PRG_HVCP3_54CB1();

PRG_HVCP3_56CB1();

END_PROGRAM

// ---- POUs/HVCP3/PRG_HVCP3_10CB1.TcPOU
PROGRAM PRG_HVCP3_10CB1
VAR
    // Function Block Instance
    fbDisconnector		: FB_DisconnectorControl;
	
	stDisconnectorIO	: ST_DisconnectorIO;
	
    
    // Başlangıç konfigürasyonu için flag
    bInitDone: BOOL := FALSE;	
END_VAR

IF NOT bInitDone THEN
	bInitDone := TRUE;
	RETURN;
END_IF

//*************************************************************************
// Ana Besleme Ayırıcısı
// +EP6-8CB1
//*************************************************************************
fbDisconnector(
    // Fiziksel Girişler
    bContactorOn_FB 	:= stDisconnectorIO.bContactorOn_FB,
    bContactorOff_FB 	:= stDisconnectorIO.bContactorOff_FB,
    bLimitOn 			:= stDisconnectorIO.bLimitOn,
    bLimitOff 			:= stDisconnectorIO.bLimitOff,
    bThermalFault 		:= stDisconnectorIO.bThermalFault,
    bEarthSwitchOn 		:= stDisconnectorIO.bEarthSwitchOn,
    bEarthSwitchOff 	:= stDisconnectorIO.bEarthSwitchOff,
    bPLCControl 		:= stDisconnectorIO.bPLCControl,
    
    // Güvenlik Girişleri
    bSafetyLoop 		:= GVL_Alarm.bSafetyLoop,
    bInterlock 			:= FALSE,
    
    // Sistem Girişleri
    bMasterReset 		:= GVL_Alarm.bMasterReset,
    
    // HMI Bağlantısı
    stHMI 				:= GVL_HVCP3.stMainDisconnectorHMI,
    
    // Fiziksel Çıkışlar
    bContactorOn_Out 	=> stDisconnectorIO.bContactorOn_Out,
    bContactorOff_Out 	=> stDisconnectorIO.bContactorOff_Out
);

METHOD M_Init : BOOL
VAR_INPUT
END_VAR

GVL_HVCP3.stMainDisconnectorHMI.stConfig.bEarthSwitchExists := TRUE;
GVL_HVCP3.stMainDisconnectorHMI.stConfig.bGrounded := TRUE;
GVL_HVCP3.stMainDisconnectorHMI.stConfig.bInterlockEnable := TRUE;
GVL_HVCP3.stMainDisconnectorHMI.stConfig.dwOperationLimit := 10000;
GVL_HVCP3.stMainDisconnectorHMI.stConfig.nPhaseCount := 3;
GVL_HVCP3.stMainDisconnectorHMI.stConfig.rRatedCurrent := 2000.0;
GVL_HVCP3.stMainDisconnectorHMI.stConfig.rRatedVoltage := 72000.0;
GVL_HVCP3.stMainDisconnectorHMI.stConfig.sProductCode := '';
GVL_HVCP3.stMainDisconnectorHMI.stConfig.sProjectCode := '+EP9-10CB1';
GVL_HVCP3.stMainDisconnectorHMI.stConfig.tContactorDelay := T#500MS;
GVL_HVCP3.stMainDisconnectorHMI.stConfig.tMotionTimeout := T#50S;
END_METHOD

END_PROGRAM

// ---- POUs/HVCP3/PRG_HVCP3_12CB1.TcPOU
PROGRAM PRG_HVCP3_12CB1
VAR
    // Function Block Instance
    fbDisconnector		: FB_DisconnectorControl;
	
	stDisconnectorIO	: ST_DisconnectorIO;
	
    
    // Başlangıç konfigürasyonu için flag
    bInitDone: BOOL := FALSE;	
END_VAR

IF NOT bInitDone THEN
	bInitDone := TRUE;
	RETURN;
END_IF

//*************************************************************************
// Ana Besleme Ayırıcısı
// +EP6-8CB1
//*************************************************************************
fbDisconnector(
    // Fiziksel Girişler
    bContactorOn_FB 	:= stDisconnectorIO.bContactorOn_FB,
    bContactorOff_FB 	:= stDisconnectorIO.bContactorOff_FB,
    bLimitOn 			:= stDisconnectorIO.bLimitOn,
    bLimitOff 			:= stDisconnectorIO.bLimitOff,
    bThermalFault 		:= stDisconnectorIO.bThermalFault,
    bEarthSwitchOn 		:= stDisconnectorIO.bEarthSwitchOn,
    bEarthSwitchOff 	:= stDisconnectorIO.bEarthSwitchOff,
    bPLCControl 		:= stDisconnectorIO.bPLCControl,
    
    // Güvenlik Girişleri
    bSafetyLoop 		:= GVL_Alarm.bSafetyLoop,
    bInterlock 			:= FALSE,
    
    // Sistem Girişleri
    bMasterReset 		:= GVL_Alarm.bMasterReset,
    
    // HMI Bağlantısı
    stHMI 				:= GVL_HVCP3.st12CB1HMI,
    
    // Fiziksel Çıkışlar
    bContactorOn_Out 	=> stDisconnectorIO.bContactorOn_Out,
    bContactorOff_Out 	=> stDisconnectorIO.bContactorOff_Out
);

METHOD M_Init : BOOL
VAR_INPUT
END_VAR

GVL_HVCP3.st12CB1HMI.stConfig.bEarthSwitchExists := FALSE;
GVL_HVCP3.st12CB1HMI.stConfig.bGrounded := FALSE;
GVL_HVCP3.st12CB1HMI.stConfig.bInterlockEnable := TRUE;
GVL_HVCP3.st12CB1HMI.stConfig.dwOperationLimit := 10000;
GVL_HVCP3.st12CB1HMI.stConfig.nPhaseCount := 3;
GVL_HVCP3.st12CB1HMI.stConfig.rRatedCurrent := 1000.0;
GVL_HVCP3.st12CB1HMI.stConfig.rRatedVoltage := 36000.0;
GVL_HVCP3.st12CB1HMI.stConfig.sProductCode := '';
GVL_HVCP3.st12CB1HMI.stConfig.sProjectCode := '+EP9-12CB1';
GVL_HVCP3.st12CB1HMI.stConfig.tContactorDelay := T#500MS;
GVL_HVCP3.st12CB1HMI.stConfig.tMotionTimeout := T#50S;
END_METHOD

END_PROGRAM

// ---- POUs/HVCP3/PRG_HVCP3_14CB1.TcPOU
PROGRAM PRG_HVCP3_14CB1
VAR
    // Function Block Instance
    fbDisconnector		: FB_DisconnectorControl;
	
	stDisconnectorIO	: ST_DisconnectorIO;
	
    
    // Başlangıç konfigürasyonu için flag
    bInitDone: BOOL := FALSE;	
END_VAR

IF NOT bInitDone THEN
	bInitDone := TRUE;
	RETURN;
END_IF

//*************************************************************************
// Ana Besleme Ayırıcısı
// +EP6-8CB1
//*************************************************************************
fbDisconnector(
    // Fiziksel Girişler
    bContactorOn_FB 	:= stDisconnectorIO.bContactorOn_FB,
    bContactorOff_FB 	:= stDisconnectorIO.bContactorOff_FB,
    bLimitOn 			:= stDisconnectorIO.bLimitOn,
    bLimitOff 			:= stDisconnectorIO.bLimitOff,
    bThermalFault 		:= stDisconnectorIO.bThermalFault,
    bEarthSwitchOn 		:= stDisconnectorIO.bEarthSwitchOn,
    bEarthSwitchOff 	:= stDisconnectorIO.bEarthSwitchOff,
    bPLCControl 		:= stDisconnectorIO.bPLCControl,
    
    // Güvenlik Girişleri
    bSafetyLoop 		:= GVL_Alarm.bSafetyLoop,
    bInterlock 			:= FALSE,
    
    // Sistem Girişleri
    bMasterReset 		:= GVL_Alarm.bMasterReset,
    
    // HMI Bağlantısı
    stHMI 				:= GVL_HVCP3.st14CB1HMI,
    
    // Fiziksel Çıkışlar
    bContactorOn_Out 	=> stDisconnectorIO.bContactorOn_Out,
    bContactorOff_Out 	=> stDisconnectorIO.bContactorOff_Out
);

METHOD M_Init : BOOL
VAR_INPUT
END_VAR

GVL_HVCP3.st14CB1HMI.stConfig.bEarthSwitchExists := FALSE;
GVL_HVCP3.st14CB1HMI.stConfig.bGrounded := FALSE;
GVL_HVCP3.st14CB1HMI.stConfig.bInterlockEnable := TRUE;
GVL_HVCP3.st14CB1HMI.stConfig.dwOperationLimit := 10000;
GVL_HVCP3.st14CB1HMI.stConfig.nPhaseCount := 3;
GVL_HVCP3.st14CB1HMI.stConfig.rRatedCurrent := 1000.0;
GVL_HVCP3.st14CB1HMI.stConfig.rRatedVoltage := 36000.0;
GVL_HVCP3.st14CB1HMI.stConfig.sProductCode := '';
GVL_HVCP3.st14CB1HMI.stConfig.sProjectCode := '+EP9-14CB1';
GVL_HVCP3.st14CB1HMI.stConfig.tContactorDelay := T#500MS;
GVL_HVCP3.st14CB1HMI.stConfig.tMotionTimeout := T#50S;
END_METHOD

END_PROGRAM

// ---- POUs/HVCP3/PRG_HVCP3_16CB1.TcPOU
PROGRAM PRG_HVCP3_16CB1
VAR
    // Function Block Instance
    fbDisconnector		: FB_DisconnectorControl;
	
	stDisconnectorIO	: ST_DisconnectorIO;
	
    
    // Başlangıç konfigürasyonu için flag
    bInitDone: BOOL := FALSE;	
END_VAR

IF NOT bInitDone THEN
	bInitDone := TRUE;
	RETURN;
END_IF

//*************************************************************************
// Ana Besleme Ayırıcısı
// +EP6-8CB1
//*************************************************************************
fbDisconnector(
    // Fiziksel Girişler
    bContactorOn_FB 	:= stDisconnectorIO.bContactorOn_FB,
    bContactorOff_FB 	:= stDisconnectorIO.bContactorOff_FB,
    bLimitOn 			:= stDisconnectorIO.bLimitOn,
    bLimitOff 			:= stDisconnectorIO.bLimitOff,
    bThermalFault 		:= stDisconnectorIO.bThermalFault,
    bEarthSwitchOn 		:= stDisconnectorIO.bEarthSwitchOn,
    bEarthSwitchOff 	:= stDisconnectorIO.bEarthSwitchOff,
    bPLCControl 		:= stDisconnectorIO.bPLCControl,
    
    // Güvenlik Girişleri
    bSafetyLoop 		:= GVL_Alarm.bSafetyLoop,
    bInterlock 			:= FALSE,
    
    // Sistem Girişleri
    bMasterReset 		:= GVL_Alarm.bMasterReset,
    
    // HMI Bağlantısı
    stHMI 				:= GVL_HVCP3.st16CB1HMI,
    
    // Fiziksel Çıkışlar
    bContactorOn_Out 	=> stDisconnectorIO.bContactorOn_Out,
    bContactorOff_Out 	=> stDisconnectorIO.bContactorOff_Out
);

METHOD M_Init : BOOL
VAR_INPUT
END_VAR

GVL_HVCP3.st16CB1HMI.stConfig.bEarthSwitchExists := FALSE;
GVL_HVCP3.st16CB1HMI.stConfig.bGrounded := FALSE;
GVL_HVCP3.st16CB1HMI.stConfig.bInterlockEnable := TRUE;
GVL_HVCP3.st16CB1HMI.stConfig.dwOperationLimit := 10000;
GVL_HVCP3.st16CB1HMI.stConfig.nPhaseCount := 3;
GVL_HVCP3.st16CB1HMI.stConfig.rRatedCurrent := 1000.0;
GVL_HVCP3.st16CB1HMI.stConfig.rRatedVoltage := 36000.0;
GVL_HVCP3.st16CB1HMI.stConfig.sProductCode := '';
GVL_HVCP3.st16CB1HMI.stConfig.sProjectCode := '+EP9-16CB1';
GVL_HVCP3.st16CB1HMI.stConfig.tContactorDelay := T#500MS;
GVL_HVCP3.st16CB1HMI.stConfig.tMotionTimeout := T#50S;
END_METHOD

END_PROGRAM

// ---- POUs/HVCP3/PRG_HVCP3_18CB1.TcPOU
PROGRAM PRG_HVCP3_18CB1
VAR
    // Function Block Instance
    fbDisconnector		: FB_DisconnectorControl;
	
	stDisconnectorIO	: ST_DisconnectorIO;
	
    
    // Başlangıç konfigürasyonu için flag
    bInitDone: BOOL := FALSE;	
END_VAR

IF NOT bInitDone THEN
	bInitDone := TRUE;
	RETURN;
END_IF

//*************************************************************************
// Ana Besleme Ayırıcısı
// +EP6-8CB1
//*************************************************************************
fbDisconnector(
    // Fiziksel Girişler
    bContactorOn_FB 	:= stDisconnectorIO.bContactorOn_FB,
    bContactorOff_FB 	:= stDisconnectorIO.bContactorOff_FB,
    bLimitOn 			:= stDisconnectorIO.bLimitOn,
    bLimitOff 			:= stDisconnectorIO.bLimitOff,
    bThermalFault 		:= stDisconnectorIO.bThermalFault,
    bEarthSwitchOn 		:= stDisconnectorIO.bEarthSwitchOn,
    bEarthSwitchOff 	:= stDisconnectorIO.bEarthSwitchOff,
    bPLCControl 		:= stDisconnectorIO.bPLCControl,
    
    // Güvenlik Girişleri
    bSafetyLoop 		:= GVL_Alarm.bSafetyLoop,
    bInterlock 			:= FALSE,
    
    // Sistem Girişleri
    bMasterReset 		:= GVL_Alarm.bMasterReset,
    
    // HMI Bağlantısı
    stHMI 				:= GVL_HVCP3.st18CB1HMI,
    
    // Fiziksel Çıkışlar
    bContactorOn_Out 	=> stDisconnectorIO.bContactorOn_Out,
    bContactorOff_Out 	=> stDisconnectorIO.bContactorOff_Out
);

METHOD M_Init : BOOL
VAR_INPUT
END_VAR

GVL_HVCP3.st18CB1HMI.stConfig.bEarthSwitchExists := FALSE;
GVL_HVCP3.st18CB1HMI.stConfig.bGrounded := FALSE;
GVL_HVCP3.st18CB1HMI.stConfig.bInterlockEnable := TRUE;
GVL_HVCP3.st18CB1HMI.stConfig.dwOperationLimit := 10000;
GVL_HVCP3.st18CB1HMI.stConfig.nPhaseCount := 3;
GVL_HVCP3.st18CB1HMI.stConfig.rRatedCurrent := 1000.0;
GVL_HVCP3.st18CB1HMI.stConfig.rRatedVoltage := 36000.0;
GVL_HVCP3.st18CB1HMI.stConfig.sProductCode := '';
GVL_HVCP3.st18CB1HMI.stConfig.sProjectCode := '+EP9-18CB1';
GVL_HVCP3.st18CB1HMI.stConfig.tContactorDelay := T#500MS;
GVL_HVCP3.st18CB1HMI.stConfig.tMotionTimeout := T#50S;
END_METHOD

END_PROGRAM

// ---- POUs/HVCP3/PRG_HVCP3_20CB1.TcPOU
PROGRAM PRG_HVCP3_20CB1
VAR
    // Function Block Instance
    fbDisconnector		: FB_DisconnectorControl;
	
	stDisconnectorIO	: ST_DisconnectorIO;
	
    
    // Başlangıç konfigürasyonu için flag
    bInitDone: BOOL := FALSE;	
END_VAR

IF NOT bInitDone THEN
	bInitDone := TRUE;
	RETURN;
END_IF

//*************************************************************************
// Ana Besleme Ayırıcısı
// +EP6-8CB1
//*************************************************************************
fbDisconnector(
    // Fiziksel Girişler
    bContactorOn_FB 	:= stDisconnectorIO.bContactorOn_FB,
    bContactorOff_FB 	:= stDisconnectorIO.bContactorOff_FB,
    bLimitOn 			:= stDisconnectorIO.bLimitOn,
    bLimitOff 			:= stDisconnectorIO.bLimitOff,
    bThermalFault 		:= stDisconnectorIO.bThermalFault,
    bEarthSwitchOn 		:= stDisconnectorIO.bEarthSwitchOn,
    bEarthSwitchOff 	:= stDisconnectorIO.bEarthSwitchOff,
    bPLCControl 		:= stDisconnectorIO.bPLCControl,
    
    // Güvenlik Girişleri
    bSafetyLoop 		:= GVL_Alarm.bSafetyLoop,
    bInterlock 			:= FALSE,
    
    // Sistem Girişleri
    bMasterReset 		:= GVL_Alarm.bMasterReset,
    
    // HMI Bağlantısı
    stHMI 				:= GVL_HVCP3.st20CB1HMI,
    
    // Fiziksel Çıkışlar
    bContactorOn_Out 	=> stDisconnectorIO.bContactorOn_Out,
    bContactorOff_Out 	=> stDisconnectorIO.bContactorOff_Out
);

METHOD M_Init : BOOL
VAR_INPUT
END_VAR

GVL_HVCP3.st20CB1HMI.stConfig.bEarthSwitchExists := FALSE;
GVL_HVCP3.st20CB1HMI.stConfig.bGrounded := FALSE;
GVL_HVCP3.st20CB1HMI.stConfig.bInterlockEnable := TRUE;
GVL_HVCP3.st20CB1HMI.stConfig.dwOperationLimit := 10000;
GVL_HVCP3.st20CB1HMI.stConfig.nPhaseCount := 3;
GVL_HVCP3.st20CB1HMI.stConfig.rRatedCurrent := 1000.0;
GVL_HVCP3.st20CB1HMI.stConfig.rRatedVoltage := 36000.0;
GVL_HVCP3.st20CB1HMI.stConfig.sProductCode := '';
GVL_HVCP3.st20CB1HMI.stConfig.sProjectCode := '+EP9-20CB1';
GVL_HVCP3.st20CB1HMI.stConfig.tContactorDelay := T#500MS;
GVL_HVCP3.st20CB1HMI.stConfig.tMotionTimeout := T#50S;
END_METHOD

END_PROGRAM

// ---- POUs/HVCP3/PRG_HVCP3_22CB1.TcPOU
PROGRAM PRG_HVCP3_22CB1
VAR
    // Function Block Instance
    fbDisconnector		: FB_DisconnectorControl;
	
	stDisconnectorIO	: ST_DisconnectorIO;
	
    
    // Başlangıç konfigürasyonu için flag
    bInitDone: BOOL := FALSE;	
END_VAR

IF NOT bInitDone THEN
	bInitDone := TRUE;
	RETURN;
END_IF

//*************************************************************************
// Ana Besleme Ayırıcısı
// +EP6-8CB1
//*************************************************************************
fbDisconnector(
    // Fiziksel Girişler
    bContactorOn_FB 	:= stDisconnectorIO.bContactorOn_FB,
    bContactorOff_FB 	:= stDisconnectorIO.bContactorOff_FB,
    bLimitOn 			:= stDisconnectorIO.bLimitOn,
    bLimitOff 			:= stDisconnectorIO.bLimitOff,
    bThermalFault 		:= stDisconnectorIO.bThermalFault,
    bEarthSwitchOn 		:= stDisconnectorIO.bEarthSwitchOn,
    bEarthSwitchOff 	:= stDisconnectorIO.bEarthSwitchOff,
    bPLCControl 		:= stDisconnectorIO.bPLCControl,
    
    // Güvenlik Girişleri
    bSafetyLoop 		:= GVL_Alarm.bSafetyLoop,
    bInterlock 			:= FALSE,
    
    // Sistem Girişleri
    bMasterReset 		:= GVL_Alarm.bMasterReset,
    
    // HMI Bağlantısı
    stHMI 				:= GVL_HVCP3.st22CB1HMI,
    
    // Fiziksel Çıkışlar
    bContactorOn_Out 	=> stDisconnectorIO.bContactorOn_Out,
    bContactorOff_Out 	=> stDisconnectorIO.bContactorOff_Out
);

METHOD M_Init : BOOL
VAR_INPUT
END_VAR

GVL_HVCP3.st22CB1HMI.stConfig.bEarthSwitchExists := FALSE;
GVL_HVCP3.st22CB1HMI.stConfig.bGrounded := FALSE;
GVL_HVCP3.st22CB1HMI.stConfig.bInterlockEnable := TRUE;
GVL_HVCP3.st22CB1HMI.stConfig.dwOperationLimit := 10000;
GVL_HVCP3.st22CB1HMI.stConfig.nPhaseCount := 3;
GVL_HVCP3.st22CB1HMI.stConfig.rRatedCurrent := 1000.0;
GVL_HVCP3.st22CB1HMI.stConfig.rRatedVoltage := 36000.0;
GVL_HVCP3.st22CB1HMI.stConfig.sProductCode := '';
GVL_HVCP3.st22CB1HMI.stConfig.sProjectCode := '+EP9-22CB1';
GVL_HVCP3.st22CB1HMI.stConfig.tContactorDelay := T#500MS;
GVL_HVCP3.st22CB1HMI.stConfig.tMotionTimeout := T#50S;
END_METHOD

END_PROGRAM

// ---- POUs/HVCP3/PRG_HVCP3_24CB1.TcPOU
PROGRAM PRG_HVCP3_24CB1
VAR
    // Function Block Instance
    fbDisconnector		: FB_DisconnectorControl;
	
	stDisconnectorIO	: ST_DisconnectorIO;
	
    
    // Başlangıç konfigürasyonu için flag
    bInitDone: BOOL := FALSE;	
END_VAR

IF NOT bInitDone THEN
	bInitDone := TRUE;
	RETURN;
END_IF

//*************************************************************************
// Ana Besleme Ayırıcısı
// +EP6-8CB1
//*************************************************************************
fbDisconnector(
    // Fiziksel Girişler
    bContactorOn_FB 	:= stDisconnectorIO.bContactorOn_FB,
    bContactorOff_FB 	:= stDisconnectorIO.bContactorOff_FB,
    bLimitOn 			:= stDisconnectorIO.bLimitOn,
    bLimitOff 			:= stDisconnectorIO.bLimitOff,
    bThermalFault 		:= stDisconnectorIO.bThermalFault,
    bEarthSwitchOn 		:= stDisconnectorIO.bEarthSwitchOn,
    bEarthSwitchOff 	:= stDisconnectorIO.bEarthSwitchOff,
    bPLCControl 		:= stDisconnectorIO.bPLCControl,
    
    // Güvenlik Girişleri
    bSafetyLoop 		:= GVL_Alarm.bSafetyLoop,
    bInterlock 			:= FALSE,
    
    // Sistem Girişleri
    bMasterReset 		:= GVL_Alarm.bMasterReset,
    
    // HMI Bağlantısı
    stHMI 				:= GVL_HVCP3.st24CB1HMI,
    
    // Fiziksel Çıkışlar
    bContactorOn_Out 	=> stDisconnectorIO.bContactorOn_Out,
    bContactorOff_Out 	=> stDisconnectorIO.bContactorOff_Out
);

METHOD M_Init : BOOL
VAR_INPUT
END_VAR

GVL_HVCP3.st16CB1HMI.stConfig.bEarthSwitchExists := FALSE;
GVL_HVCP3.st16CB1HMI.stConfig.bGrounded := FALSE;
GVL_HVCP3.st16CB1HMI.stConfig.bInterlockEnable := TRUE;
GVL_HVCP3.st16CB1HMI.stConfig.dwOperationLimit := 10000;
GVL_HVCP3.st16CB1HMI.stConfig.nPhaseCount := 3;
GVL_HVCP3.st16CB1HMI.stConfig.rRatedCurrent := 1000.0;
GVL_HVCP3.st16CB1HMI.stConfig.rRatedVoltage := 36000.0;
GVL_HVCP3.st16CB1HMI.stConfig.sProductCode := '';
GVL_HVCP3.st16CB1HMI.stConfig.sProjectCode := '+EP9-24CB1';
GVL_HVCP3.st16CB1HMI.stConfig.tContactorDelay := T#500MS;
GVL_HVCP3.st16CB1HMI.stConfig.tMotionTimeout := T#50S;
END_METHOD

END_PROGRAM

// ---- POUs/HVCP3/PRG_HVCP3_26CB1.TcPOU
PROGRAM PRG_HVCP3_26CB1
VAR
    // Function Block Instance
    fbDisconnector		: FB_DisconnectorControl;
	
	stDisconnectorIO	: ST_DisconnectorIO;
	
    
    // Başlangıç konfigürasyonu için flag
    bInitDone: BOOL := FALSE;	
END_VAR

IF NOT bInitDone THEN
	bInitDone := TRUE;
	RETURN;
END_IF

//*************************************************************************
// Ana Besleme Ayırıcısı
// +EP6-8CB1
//*************************************************************************
fbDisconnector(
    // Fiziksel Girişler
    bContactorOn_FB 	:= stDisconnectorIO.bContactorOn_FB,
    bContactorOff_FB 	:= stDisconnectorIO.bContactorOff_FB,
    bLimitOn 			:= stDisconnectorIO.bLimitOn,
    bLimitOff 			:= stDisconnectorIO.bLimitOff,
    bThermalFault 		:= stDisconnectorIO.bThermalFault,
    bEarthSwitchOn 		:= stDisconnectorIO.bEarthSwitchOn,
    bEarthSwitchOff 	:= stDisconnectorIO.bEarthSwitchOff,
    bPLCControl 		:= stDisconnectorIO.bPLCControl,
    
    // Güvenlik Girişleri
    bSafetyLoop 		:= GVL_Alarm.bSafetyLoop,
    bInterlock 			:= FALSE,
    
    // Sistem Girişleri
    bMasterReset 		:= GVL_Alarm.bMasterReset,
    
    // HMI Bağlantısı
    stHMI 				:= GVL_HVCP3.st26CB1HMI,
    
    // Fiziksel Çıkışlar
    bContactorOn_Out 	=> stDisconnectorIO.bContactorOn_Out,
    bContactorOff_Out 	=> stDisconnectorIO.bContactorOff_Out
);

METHOD M_Init : BOOL
VAR_INPUT
END_VAR

GVL_HVCP3.st16CB1HMI.stConfig.bEarthSwitchExists := FALSE;
GVL_HVCP3.st16CB1HMI.stConfig.bGrounded := FALSE;
GVL_HVCP3.st16CB1HMI.stConfig.bInterlockEnable := TRUE;
GVL_HVCP3.st16CB1HMI.stConfig.dwOperationLimit := 10000;
GVL_HVCP3.st16CB1HMI.stConfig.nPhaseCount := 3;
GVL_HVCP3.st16CB1HMI.stConfig.rRatedCurrent := 1000.0;
GVL_HVCP3.st16CB1HMI.stConfig.rRatedVoltage := 36000.0;
GVL_HVCP3.st16CB1HMI.stConfig.sProductCode := '';
GVL_HVCP3.st16CB1HMI.stConfig.sProjectCode := '+EP9-26CB1';
GVL_HVCP3.st16CB1HMI.stConfig.tContactorDelay := T#500MS;
GVL_HVCP3.st16CB1HMI.stConfig.tMotionTimeout := T#50S;
END_METHOD

END_PROGRAM

// ---- POUs/HVCP3/PRG_HVCP3_28CB1.TcPOU
PROGRAM PRG_HVCP3_28CB1
VAR
    // Function Block Instance
    fbDisconnector		: FB_DisconnectorControl;
	
	stDisconnectorIO	: ST_DisconnectorIO;
	
    
    // Başlangıç konfigürasyonu için flag
    bInitDone: BOOL := FALSE;	
END_VAR

IF NOT bInitDone THEN
	bInitDone := TRUE;
	RETURN;
END_IF

//*************************************************************************
// Ana Besleme Ayırıcısı
// +EP6-8CB1
//*************************************************************************
fbDisconnector(
    // Fiziksel Girişler
    bContactorOn_FB 	:= stDisconnectorIO.bContactorOn_FB,
    bContactorOff_FB 	:= stDisconnectorIO.bContactorOff_FB,
    bLimitOn 			:= stDisconnectorIO.bLimitOn,
    bLimitOff 			:= stDisconnectorIO.bLimitOff,
    bThermalFault 		:= stDisconnectorIO.bThermalFault,
    bEarthSwitchOn 		:= stDisconnectorIO.bEarthSwitchOn,
    bEarthSwitchOff 	:= stDisconnectorIO.bEarthSwitchOff,
    bPLCControl 		:= stDisconnectorIO.bPLCControl,
    
    // Güvenlik Girişleri
    bSafetyLoop 		:= GVL_Alarm.bSafetyLoop,
    bInterlock 			:= FALSE,
    
    // Sistem Girişleri
    bMasterReset 		:= GVL_Alarm.bMasterReset,
    
    // HMI Bağlantısı
    stHMI 				:= GVL_HVCP3.st28CB1HMI,
    
    // Fiziksel Çıkışlar
    bContactorOn_Out 	=> stDisconnectorIO.bContactorOn_Out,
    bContactorOff_Out 	=> stDisconnectorIO.bContactorOff_Out
);

METHOD M_Init : BOOL
VAR_INPUT
END_VAR

GVL_HVCP3.st16CB1HMI.stConfig.bEarthSwitchExists := FALSE;
GVL_HVCP3.st16CB1HMI.stConfig.bGrounded := FALSE;
GVL_HVCP3.st16CB1HMI.stConfig.bInterlockEnable := TRUE;
GVL_HVCP3.st16CB1HMI.stConfig.dwOperationLimit := 10000;
GVL_HVCP3.st16CB1HMI.stConfig.nPhaseCount := 3;
GVL_HVCP3.st16CB1HMI.stConfig.rRatedCurrent := 1000.0;
GVL_HVCP3.st16CB1HMI.stConfig.rRatedVoltage := 36000.0;
GVL_HVCP3.st16CB1HMI.stConfig.sProductCode := '';
GVL_HVCP3.st16CB1HMI.stConfig.sProjectCode := '+EP9-28CB1';
GVL_HVCP3.st16CB1HMI.stConfig.tContactorDelay := T#500MS;
GVL_HVCP3.st16CB1HMI.stConfig.tMotionTimeout := T#50S;
END_METHOD

END_PROGRAM

// ---- POUs/HVCP3/PRG_HVCP3_30CB1.TcPOU
PROGRAM PRG_HVCP3_30CB1
VAR
    // Function Block Instance
    fbDisconnector		: FB_DisconnectorControl;
	
	stDisconnectorIO	: ST_DisconnectorIO;
	
    
    // Başlangıç konfigürasyonu için flag
    bInitDone: BOOL := FALSE;	
END_VAR

IF NOT bInitDone THEN
	bInitDone := TRUE;
	RETURN;
END_IF

//*************************************************************************
// Ana Besleme Ayırıcısı
// +EP6-8CB1
//*************************************************************************
fbDisconnector(
    // Fiziksel Girişler
    bContactorOn_FB 	:= stDisconnectorIO.bContactorOn_FB,
    bContactorOff_FB 	:= stDisconnectorIO.bContactorOff_FB,
    bLimitOn 			:= stDisconnectorIO.bLimitOn,
    bLimitOff 			:= stDisconnectorIO.bLimitOff,
    bThermalFault 		:= stDisconnectorIO.bThermalFault,
    bEarthSwitchOn 		:= stDisconnectorIO.bEarthSwitchOn,
    bEarthSwitchOff 	:= stDisconnectorIO.bEarthSwitchOff,
    bPLCControl 		:= stDisconnectorIO.bPLCControl,
    
    // Güvenlik Girişleri
    bSafetyLoop 		:= GVL_Alarm.bSafetyLoop,
    bInterlock 			:= FALSE,
    
    // Sistem Girişleri
    bMasterReset 		:= GVL_Alarm.bMasterReset,
    
    // HMI Bağlantısı
    stHMI 				:= GVL_HVCP3.st30CB1HMI,
    
    // Fiziksel Çıkışlar
    bContactorOn_Out 	=> stDisconnectorIO.bContactorOn_Out,
    bContactorOff_Out 	=> stDisconnectorIO.bContactorOff_Out
);

METHOD M_Init : BOOL
VAR_INPUT
END_VAR

GVL_HVCP3.st16CB1HMI.stConfig.bEarthSwitchExists := FALSE;
GVL_HVCP3.st16CB1HMI.stConfig.bGrounded := FALSE;
GVL_HVCP3.st16CB1HMI.stConfig.bInterlockEnable := TRUE;
GVL_HVCP3.st16CB1HMI.stConfig.dwOperationLimit := 10000;
GVL_HVCP3.st16CB1HMI.stConfig.nPhaseCount := 3;
GVL_HVCP3.st16CB1HMI.stConfig.rRatedCurrent := 1000.0;
GVL_HVCP3.st16CB1HMI.stConfig.rRatedVoltage := 36000.0;
GVL_HVCP3.st16CB1HMI.stConfig.sProductCode := '';
GVL_HVCP3.st16CB1HMI.stConfig.sProjectCode := '+EP9-30CB1';
GVL_HVCP3.st16CB1HMI.stConfig.tContactorDelay := T#500MS;
GVL_HVCP3.st16CB1HMI.stConfig.tMotionTimeout := T#50S;
END_METHOD

END_PROGRAM

// ---- POUs/HVCP3/PRG_HVCP3_32CB1.TcPOU
PROGRAM PRG_HVCP3_32CB1
VAR
    // Function Block Instance
    fbDisconnector		: FB_DisconnectorControl;
	
	stDisconnectorIO	: ST_DisconnectorIO;
	
    
    // Başlangıç konfigürasyonu için flag
    bInitDone: BOOL := FALSE;	
END_VAR

IF NOT bInitDone THEN
	bInitDone := TRUE;
	RETURN;
END_IF

//*************************************************************************
// Ana Besleme Ayırıcısı
// +EP6-8CB1
//*************************************************************************
fbDisconnector(
    // Fiziksel Girişler
    bContactorOn_FB 	:= stDisconnectorIO.bContactorOn_FB,
    bContactorOff_FB 	:= stDisconnectorIO.bContactorOff_FB,
    bLimitOn 			:= stDisconnectorIO.bLimitOn,
    bLimitOff 			:= stDisconnectorIO.bLimitOff,
    bThermalFault 		:= stDisconnectorIO.bThermalFault,
    bEarthSwitchOn 		:= stDisconnectorIO.bEarthSwitchOn,
    bEarthSwitchOff 	:= stDisconnectorIO.bEarthSwitchOff,
    bPLCControl 		:= stDisconnectorIO.bPLCControl,
    
    // Güvenlik Girişleri
    bSafetyLoop 		:= GVL_Alarm.bSafetyLoop,
    bInterlock 			:= FALSE,
    
    // Sistem Girişleri
    bMasterReset 		:= GVL_Alarm.bMasterReset,
    
    // HMI Bağlantısı
    stHMI 				:= GVL_HVCP3.st32CB1HMI,
    
    // Fiziksel Çıkışlar
    bContactorOn_Out 	=> stDisconnectorIO.bContactorOn_Out,
    bContactorOff_Out 	=> stDisconnectorIO.bContactorOff_Out
);

METHOD M_Init : BOOL
VAR_INPUT
END_VAR

GVL_HVCP3.st16CB1HMI.stConfig.bEarthSwitchExists := FALSE;
GVL_HVCP3.st16CB1HMI.stConfig.bGrounded := FALSE;
GVL_HVCP3.st16CB1HMI.stConfig.bInterlockEnable := TRUE;
GVL_HVCP3.st16CB1HMI.stConfig.dwOperationLimit := 10000;
GVL_HVCP3.st16CB1HMI.stConfig.nPhaseCount := 3;
GVL_HVCP3.st16CB1HMI.stConfig.rRatedCurrent := 1000.0;
GVL_HVCP3.st16CB1HMI.stConfig.rRatedVoltage := 36000.0;
GVL_HVCP3.st16CB1HMI.stConfig.sProductCode := '';
GVL_HVCP3.st16CB1HMI.stConfig.sProjectCode := '+EP9-32CB1';
GVL_HVCP3.st16CB1HMI.stConfig.tContactorDelay := T#500MS;
GVL_HVCP3.st16CB1HMI.stConfig.tMotionTimeout := T#50S;
END_METHOD

END_PROGRAM

// ---- POUs/HVCP3/PRG_HVCP3_34CB1.TcPOU
PROGRAM PRG_HVCP3_34CB1
VAR
    // Function Block Instance
    fbDisconnector		: FB_DisconnectorControl;
	
	stDisconnectorIO	: ST_DisconnectorIO;
	
    
    // Başlangıç konfigürasyonu için flag
    bInitDone: BOOL := FALSE;	
END_VAR

IF NOT bInitDone THEN
	bInitDone := TRUE;
	RETURN;
END_IF

//*************************************************************************
// Ana Besleme Ayırıcısı
// +EP6-8CB1
//*************************************************************************
fbDisconnector(
    // Fiziksel Girişler
    bContactorOn_FB 	:= stDisconnectorIO.bContactorOn_FB,
    bContactorOff_FB 	:= stDisconnectorIO.bContactorOff_FB,
    bLimitOn 			:= stDisconnectorIO.bLimitOn,
    bLimitOff 			:= stDisconnectorIO.bLimitOff,
    bThermalFault 		:= stDisconnectorIO.bThermalFault,
    bEarthSwitchOn 		:= stDisconnectorIO.bEarthSwitchOn,
    bEarthSwitchOff 	:= stDisconnectorIO.bEarthSwitchOff,
    bPLCControl 		:= stDisconnectorIO.bPLCControl,
    
    // Güvenlik Girişleri
    bSafetyLoop 		:= GVL_Alarm.bSafetyLoop,
    bInterlock 			:= FALSE,
    
    // Sistem Girişleri
    bMasterReset 		:= GVL_Alarm.bMasterReset,
    
    // HMI Bağlantısı
    stHMI 				:= GVL_HVCP3.st34CB1HMI,
    
    // Fiziksel Çıkışlar
    bContactorOn_Out 	=> stDisconnectorIO.bContactorOn_Out,
    bContactorOff_Out 	=> stDisconnectorIO.bContactorOff_Out
);

METHOD M_Init : BOOL
VAR_INPUT
END_VAR

GVL_HVCP3.st16CB1HMI.stConfig.bEarthSwitchExists := FALSE;
GVL_HVCP3.st16CB1HMI.stConfig.bGrounded := FALSE;
GVL_HVCP3.st16CB1HMI.stConfig.bInterlockEnable := TRUE;
GVL_HVCP3.st16CB1HMI.stConfig.dwOperationLimit := 10000;
GVL_HVCP3.st16CB1HMI.stConfig.nPhaseCount := 3;
GVL_HVCP3.st16CB1HMI.stConfig.rRatedCurrent := 1000.0;
GVL_HVCP3.st16CB1HMI.stConfig.rRatedVoltage := 36000.0;
GVL_HVCP3.st16CB1HMI.stConfig.sProductCode := '';
GVL_HVCP3.st16CB1HMI.stConfig.sProjectCode := '+EP9-34CB1';
GVL_HVCP3.st16CB1HMI.stConfig.tContactorDelay := T#500MS;
GVL_HVCP3.st16CB1HMI.stConfig.tMotionTimeout := T#50S;
END_METHOD

END_PROGRAM

// ---- POUs/HVCP3/PRG_HVCP3_36CB1.TcPOU
PROGRAM PRG_HVCP3_36CB1
VAR
    // Function Block Instance
    fbDisconnector		: FB_DisconnectorControl;
	
	stDisconnectorIO	: ST_DisconnectorIO;
	
    
    // Başlangıç konfigürasyonu için flag
    bInitDone: BOOL := FALSE;	
END_VAR

IF NOT bInitDone THEN
	bInitDone := TRUE;
	RETURN;
END_IF

//*************************************************************************
// Ana Besleme Ayırıcısı
// +EP6-8CB1
//*************************************************************************
fbDisconnector(
    // Fiziksel Girişler
    bContactorOn_FB 	:= stDisconnectorIO.bContactorOn_FB,
    bContactorOff_FB 	:= stDisconnectorIO.bContactorOff_FB,
    bLimitOn 			:= stDisconnectorIO.bLimitOn,
    bLimitOff 			:= stDisconnectorIO.bLimitOff,
    bThermalFault 		:= stDisconnectorIO.bThermalFault,
    bEarthSwitchOn 		:= stDisconnectorIO.bEarthSwitchOn,
    bEarthSwitchOff 	:= stDisconnectorIO.bEarthSwitchOff,
    bPLCControl 		:= stDisconnectorIO.bPLCControl,
    
    // Güvenlik Girişleri
    bSafetyLoop 		:= GVL_Alarm.bSafetyLoop,
    bInterlock 			:= FALSE,
    
    // Sistem Girişleri
    bMasterReset 		:= GVL_Alarm.bMasterReset,
    
    // HMI Bağlantısı
    stHMI 				:= GVL_HVCP3.st36CB1HMI,
    
    // Fiziksel Çıkışlar
    bContactorOn_Out 	=> stDisconnectorIO.bContactorOn_Out,
    bContactorOff_Out 	=> stDisconnectorIO.bContactorOff_Out
);

METHOD M_Init : BOOL
VAR_INPUT
END_VAR

GVL_HVCP3.st16CB1HMI.stConfig.bEarthSwitchExists := FALSE;
GVL_HVCP3.st16CB1HMI.stConfig.bGrounded := FALSE;
GVL_HVCP3.st16CB1HMI.stConfig.bInterlockEnable := TRUE;
GVL_HVCP3.st16CB1HMI.stConfig.dwOperationLimit := 10000;
GVL_HVCP3.st16CB1HMI.stConfig.nPhaseCount := 3;
GVL_HVCP3.st16CB1HMI.stConfig.rRatedCurrent := 1000.0;
GVL_HVCP3.st16CB1HMI.stConfig.rRatedVoltage := 36000.0;
GVL_HVCP3.st16CB1HMI.stConfig.sProductCode := '';
GVL_HVCP3.st16CB1HMI.stConfig.sProjectCode := '+EP9-12CB1';
GVL_HVCP3.st16CB1HMI.stConfig.tContactorDelay := T#500MS;
GVL_HVCP3.st16CB1HMI.stConfig.tMotionTimeout := T#50S;
END_METHOD

END_PROGRAM

// ---- POUs/HVCP3/PRG_HVCP3_38CB1.TcPOU
PROGRAM PRG_HVCP3_38CB1
VAR
    // Function Block Instance
    fbDisconnector		: FB_DisconnectorControl;
	
	stDisconnectorIO	: ST_DisconnectorIO;
	
    
    // Başlangıç konfigürasyonu için flag
    bInitDone: BOOL := FALSE;	
END_VAR

IF NOT bInitDone THEN
	bInitDone := TRUE;
	RETURN;
END_IF

//*************************************************************************
// Ana Besleme Ayırıcısı
// +EP6-8CB1
//*************************************************************************
fbDisconnector(
    // Fiziksel Girişler
    bContactorOn_FB 	:= stDisconnectorIO.bContactorOn_FB,
    bContactorOff_FB 	:= stDisconnectorIO.bContactorOff_FB,
    bLimitOn 			:= stDisconnectorIO.bLimitOn,
    bLimitOff 			:= stDisconnectorIO.bLimitOff,
    bThermalFault 		:= stDisconnectorIO.bThermalFault,
    bEarthSwitchOn 		:= stDisconnectorIO.bEarthSwitchOn,
    bEarthSwitchOff 	:= stDisconnectorIO.bEarthSwitchOff,
    bPLCControl 		:= stDisconnectorIO.bPLCControl,
    
    // Güvenlik Girişleri
    bSafetyLoop 		:= GVL_Alarm.bSafetyLoop,
    bInterlock 			:= FALSE,
    
    // Sistem Girişleri
    bMasterReset 		:= GVL_Alarm.bMasterReset,
    
    // HMI Bağlantısı
    stHMI 				:= GVL_HVCP3.st38CB1HMI,
    
    // Fiziksel Çıkışlar
    bContactorOn_Out 	=> stDisconnectorIO.bContactorOn_Out,
    bContactorOff_Out 	=> stDisconnectorIO.bContactorOff_Out
);

METHOD M_Init : BOOL
VAR_INPUT
END_VAR

GVL_HVCP3.st16CB1HMI.stConfig.bEarthSwitchExists := FALSE;
GVL_HVCP3.st16CB1HMI.stConfig.bGrounded := FALSE;
GVL_HVCP3.st16CB1HMI.stConfig.bInterlockEnable := TRUE;
GVL_HVCP3.st16CB1HMI.stConfig.dwOperationLimit := 10000;
GVL_HVCP3.st16CB1HMI.stConfig.nPhaseCount := 3;
GVL_HVCP3.st16CB1HMI.stConfig.rRatedCurrent := 1000.0;
GVL_HVCP3.st16CB1HMI.stConfig.rRatedVoltage := 36000.0;
GVL_HVCP3.st16CB1HMI.stConfig.sProductCode := '';
GVL_HVCP3.st16CB1HMI.stConfig.sProjectCode := '+EP9-38CB1';
GVL_HVCP3.st16CB1HMI.stConfig.tContactorDelay := T#500MS;
GVL_HVCP3.st16CB1HMI.stConfig.tMotionTimeout := T#50S;
END_METHOD

END_PROGRAM

// ---- POUs/HVCP3/PRG_HVCP3_40CB1.TcPOU
PROGRAM PRG_HVCP3_40CB1
VAR
    // Function Block Instance
    fbDisconnector		: FB_DisconnectorControl;
	
	stDisconnectorIO	: ST_DisconnectorIO;
	
    
    // Başlangıç konfigürasyonu için flag
    bInitDone: BOOL := FALSE;	
END_VAR

IF NOT bInitDone THEN
	bInitDone := TRUE;
	RETURN;
END_IF

//*************************************************************************
// Ana Besleme Ayırıcısı
// +EP6-8CB1
//*************************************************************************
fbDisconnector(
    // Fiziksel Girişler
    bContactorOn_FB 	:= stDisconnectorIO.bContactorOn_FB,
    bContactorOff_FB 	:= stDisconnectorIO.bContactorOff_FB,
    bLimitOn 			:= stDisconnectorIO.bLimitOn,
    bLimitOff 			:= stDisconnectorIO.bLimitOff,
    bThermalFault 		:= stDisconnectorIO.bThermalFault,
    bEarthSwitchOn 		:= stDisconnectorIO.bEarthSwitchOn,
    bEarthSwitchOff 	:= stDisconnectorIO.bEarthSwitchOff,
    bPLCControl 		:= stDisconnectorIO.bPLCControl,
    
    // Güvenlik Girişleri
    bSafetyLoop 		:= GVL_Alarm.bSafetyLoop,
    bInterlock 			:= FALSE,
    
    // Sistem Girişleri
    bMasterReset 		:= GVL_Alarm.bMasterReset,
    
    // HMI Bağlantısı
    stHMI 				:= GVL_HVCP3.st40CB1HMI,
    
    // Fiziksel Çıkışlar
    bContactorOn_Out 	=> stDisconnectorIO.bContactorOn_Out,
    bContactorOff_Out 	=> stDisconnectorIO.bContactorOff_Out
);

METHOD M_Init : BOOL
VAR_INPUT
END_VAR

GVL_HVCP3.st16CB1HMI.stConfig.bEarthSwitchExists := FALSE;
GVL_HVCP3.st16CB1HMI.stConfig.bGrounded := FALSE;
GVL_HVCP3.st16CB1HMI.stConfig.bInterlockEnable := TRUE;
GVL_HVCP3.st16CB1HMI.stConfig.dwOperationLimit := 10000;
GVL_HVCP3.st16CB1HMI.stConfig.nPhaseCount := 3;
GVL_HVCP3.st16CB1HMI.stConfig.rRatedCurrent := 1000.0;
GVL_HVCP3.st16CB1HMI.stConfig.rRatedVoltage := 36000.0;
GVL_HVCP3.st16CB1HMI.stConfig.sProductCode := '';
GVL_HVCP3.st16CB1HMI.stConfig.sProjectCode := '+EP9-40CB1';
GVL_HVCP3.st16CB1HMI.stConfig.tContactorDelay := T#500MS;
GVL_HVCP3.st16CB1HMI.stConfig.tMotionTimeout := T#50S;
END_METHOD

END_PROGRAM

// ---- POUs/HVCP3/PRG_HVCP3_42CB1.TcPOU
PROGRAM PRG_HVCP3_42CB1
VAR
    // Function Block Instance
    fbDisconnector		: FB_DisconnectorControl;
	
	stDisconnectorIO	: ST_DisconnectorIO;
	
    
    // Başlangıç konfigürasyonu için flag
    bInitDone: BOOL := FALSE;	
END_VAR

IF NOT bInitDone THEN
	bInitDone := TRUE;
	RETURN;
END_IF

//*************************************************************************
// Ana Besleme Ayırıcısı
// +EP6-8CB1
//*************************************************************************
fbDisconnector(
    // Fiziksel Girişler
    bContactorOn_FB 	:= stDisconnectorIO.bContactorOn_FB,
    bContactorOff_FB 	:= stDisconnectorIO.bContactorOff_FB,
    bLimitOn 			:= stDisconnectorIO.bLimitOn,
    bLimitOff 			:= stDisconnectorIO.bLimitOff,
    bThermalFault 		:= stDisconnectorIO.bThermalFault,
    bEarthSwitchOn 		:= stDisconnectorIO.bEarthSwitchOn,
    bEarthSwitchOff 	:= stDisconnectorIO.bEarthSwitchOff,
    bPLCControl 		:= stDisconnectorIO.bPLCControl,
    
    // Güvenlik Girişleri
    bSafetyLoop 		:= GVL_Alarm.bSafetyLoop,
    bInterlock 			:= FALSE,
    
    // Sistem Girişleri
    bMasterReset 		:= GVL_Alarm.bMasterReset,
    
    // HMI Bağlantısı
    stHMI 				:= GVL_HVCP3.st42CB1HMI,
    
    // Fiziksel Çıkışlar
    bContactorOn_Out 	=> stDisconnectorIO.bContactorOn_Out,
    bContactorOff_Out 	=> stDisconnectorIO.bContactorOff_Out
);

METHOD M_Init : BOOL
VAR_INPUT
END_VAR

GVL_HVCP3.st16CB1HMI.stConfig.bEarthSwitchExists := FALSE;
GVL_HVCP3.st16CB1HMI.stConfig.bGrounded := FALSE;
GVL_HVCP3.st16CB1HMI.stConfig.bInterlockEnable := TRUE;
GVL_HVCP3.st16CB1HMI.stConfig.dwOperationLimit := 10000;
GVL_HVCP3.st16CB1HMI.stConfig.nPhaseCount := 3;
GVL_HVCP3.st16CB1HMI.stConfig.rRatedCurrent := 1000.0;
GVL_HVCP3.st16CB1HMI.stConfig.rRatedVoltage := 36000.0;
GVL_HVCP3.st16CB1HMI.stConfig.sProductCode := '';
GVL_HVCP3.st16CB1HMI.stConfig.sProjectCode := '+EP9-42CB1';
GVL_HVCP3.st16CB1HMI.stConfig.tContactorDelay := T#500MS;
GVL_HVCP3.st16CB1HMI.stConfig.tMotionTimeout := T#50S;
END_METHOD

END_PROGRAM

// ---- POUs/HVCP3/PRG_HVCP3_44CB1.TcPOU
PROGRAM PRG_HVCP3_44CB1
VAR
    // Function Block Instance
    fbDisconnector		: FB_DisconnectorControl;
	
	stDisconnectorIO	: ST_DisconnectorIO;
	
    
    // Başlangıç konfigürasyonu için flag
    bInitDone: BOOL := FALSE;	
END_VAR

IF NOT bInitDone THEN
	bInitDone := TRUE;
	RETURN;
END_IF

//*************************************************************************
// Ana Besleme Ayırıcısı
// +EP6-8CB1
//*************************************************************************
fbDisconnector(
    // Fiziksel Girişler
    bContactorOn_FB 	:= stDisconnectorIO.bContactorOn_FB,
    bContactorOff_FB 	:= stDisconnectorIO.bContactorOff_FB,
    bLimitOn 			:= stDisconnectorIO.bLimitOn,
    bLimitOff 			:= stDisconnectorIO.bLimitOff,
    bThermalFault 		:= stDisconnectorIO.bThermalFault,
    bEarthSwitchOn 		:= stDisconnectorIO.bEarthSwitchOn,
    bEarthSwitchOff 	:= stDisconnectorIO.bEarthSwitchOff,
    bPLCControl 		:= stDisconnectorIO.bPLCControl,
    
    // Güvenlik Girişleri
    bSafetyLoop 		:= GVL_Alarm.bSafetyLoop,
    bInterlock 			:= FALSE,
    
    // Sistem Girişleri
    bMasterReset 		:= GVL_Alarm.bMasterReset,
    
    // HMI Bağlantısı
    stHMI 				:= GVL_HVCP3.st44CB1HMI,
    
    // Fiziksel Çıkışlar
    bContactorOn_Out 	=> stDisconnectorIO.bContactorOn_Out,
    bContactorOff_Out 	=> stDisconnectorIO.bContactorOff_Out
);

METHOD M_Init : BOOL
VAR_INPUT
END_VAR

GVL_HVCP3.st16CB1HMI.stConfig.bEarthSwitchExists := FALSE;
GVL_HVCP3.st16CB1HMI.stConfig.bGrounded := FALSE;
GVL_HVCP3.st16CB1HMI.stConfig.bInterlockEnable := TRUE;
GVL_HVCP3.st16CB1HMI.stConfig.dwOperationLimit := 10000;
GVL_HVCP3.st16CB1HMI.stConfig.nPhaseCount := 3;
GVL_HVCP3.st16CB1HMI.stConfig.rRatedCurrent := 1000.0;
GVL_HVCP3.st16CB1HMI.stConfig.rRatedVoltage := 36000.0;
GVL_HVCP3.st16CB1HMI.stConfig.sProductCode := '';
GVL_HVCP3.st16CB1HMI.stConfig.sProjectCode := '+EP9-44CB1';
GVL_HVCP3.st16CB1HMI.stConfig.tContactorDelay := T#500MS;
GVL_HVCP3.st16CB1HMI.stConfig.tMotionTimeout := T#50S;
END_METHOD

END_PROGRAM

// ---- POUs/HVCP3/PRG_HVCP3_46CB1.TcPOU
PROGRAM PRG_HVCP3_46CB1
VAR
    // Function Block Instance
    fbDisconnector		: FB_DisconnectorControl;
	
	stDisconnectorIO	: ST_DisconnectorIO;
	
    
    // Başlangıç konfigürasyonu için flag
    bInitDone: BOOL := FALSE;	
END_VAR

IF NOT bInitDone THEN
	bInitDone := TRUE;
	RETURN;
END_IF

//*************************************************************************
// Ana Besleme Ayırıcısı
// +EP6-8CB1
//*************************************************************************
fbDisconnector(
    // Fiziksel Girişler
    bContactorOn_FB 	:= stDisconnectorIO.bContactorOn_FB,
    bContactorOff_FB 	:= stDisconnectorIO.bContactorOff_FB,
    bLimitOn 			:= stDisconnectorIO.bLimitOn,
    bLimitOff 			:= stDisconnectorIO.bLimitOff,
    bThermalFault 		:= stDisconnectorIO.bThermalFault,
    bEarthSwitchOn 		:= stDisconnectorIO.bEarthSwitchOn,
    bEarthSwitchOff 	:= stDisconnectorIO.bEarthSwitchOff,
    bPLCControl 		:= stDisconnectorIO.bPLCControl,
    
    // Güvenlik Girişleri
    bSafetyLoop 		:= GVL_Alarm.bSafetyLoop,
    bInterlock 			:= FALSE,
    
    // Sistem Girişleri
    bMasterReset 		:= GVL_Alarm.bMasterReset,
    
    // HMI Bağlantısı
    stHMI 				:= GVL_HVCP3.st46CB1HMI,
    
    // Fiziksel Çıkışlar
    bContactorOn_Out 	=> stDisconnectorIO.bContactorOn_Out,
    bContactorOff_Out 	=> stDisconnectorIO.bContactorOff_Out
);

METHOD M_Init : BOOL
VAR_INPUT
END_VAR

GVL_HVCP3.st16CB1HMI.stConfig.bEarthSwitchExists := FALSE;
GVL_HVCP3.st16CB1HMI.stConfig.bGrounded := FALSE;
GVL_HVCP3.st16CB1HMI.stConfig.bInterlockEnable := TRUE;
GVL_HVCP3.st16CB1HMI.stConfig.dwOperationLimit := 10000;
GVL_HVCP3.st16CB1HMI.stConfig.nPhaseCount := 3;
GVL_HVCP3.st16CB1HMI.stConfig.rRatedCurrent := 1000.0;
GVL_HVCP3.st16CB1HMI.stConfig.rRatedVoltage := 36000.0;
GVL_HVCP3.st16CB1HMI.stConfig.sProductCode := '';
GVL_HVCP3.st16CB1HMI.stConfig.sProjectCode := '+EP9-46CB1';
GVL_HVCP3.st16CB1HMI.stConfig.tContactorDelay := T#500MS;
GVL_HVCP3.st16CB1HMI.stConfig.tMotionTimeout := T#50S;
END_METHOD

END_PROGRAM

// ---- POUs/HVCP3/PRG_HVCP3_48CB1.TcPOU
PROGRAM PRG_HVCP3_48CB1
VAR
    // Function Block Instance
    fbDisconnector		: FB_DisconnectorControl;
	
	stDisconnectorIO	: ST_DisconnectorIO;
	
    
    // Başlangıç konfigürasyonu için flag
    bInitDone: BOOL := FALSE;	
END_VAR

IF NOT bInitDone THEN
	bInitDone := TRUE;
	RETURN;
END_IF

//*************************************************************************
// Ana Besleme Ayırıcısı
// +EP6-8CB1
//*************************************************************************
fbDisconnector(
    // Fiziksel Girişler
    bContactorOn_FB 	:= stDisconnectorIO.bContactorOn_FB,
    bContactorOff_FB 	:= stDisconnectorIO.bContactorOff_FB,
    bLimitOn 			:= stDisconnectorIO.bLimitOn,
    bLimitOff 			:= stDisconnectorIO.bLimitOff,
    bThermalFault 		:= stDisconnectorIO.bThermalFault,
    bEarthSwitchOn 		:= stDisconnectorIO.bEarthSwitchOn,
    bEarthSwitchOff 	:= stDisconnectorIO.bEarthSwitchOff,
    bPLCControl 		:= stDisconnectorIO.bPLCControl,
    
    // Güvenlik Girişleri
    bSafetyLoop 		:= GVL_Alarm.bSafetyLoop,
    bInterlock 			:= FALSE,
    
    // Sistem Girişleri
    bMasterReset 		:= GVL_Alarm.bMasterReset,
    
    // HMI Bağlantısı
    stHMI 				:= GVL_HVCP3.st48CB1HMI,
    
    // Fiziksel Çıkışlar
    bContactorOn_Out 	=> stDisconnectorIO.bContactorOn_Out,
    bContactorOff_Out 	=> stDisconnectorIO.bContactorOff_Out
);

METHOD M_Init : BOOL
VAR_INPUT
END_VAR

GVL_HVCP3.st16CB1HMI.stConfig.bEarthSwitchExists := FALSE;
GVL_HVCP3.st16CB1HMI.stConfig.bGrounded := FALSE;
GVL_HVCP3.st16CB1HMI.stConfig.bInterlockEnable := TRUE;
GVL_HVCP3.st16CB1HMI.stConfig.dwOperationLimit := 10000;
GVL_HVCP3.st16CB1HMI.stConfig.nPhaseCount := 3;
GVL_HVCP3.st16CB1HMI.stConfig.rRatedCurrent := 1000.0;
GVL_HVCP3.st16CB1HMI.stConfig.rRatedVoltage := 36000.0;
GVL_HVCP3.st16CB1HMI.stConfig.sProductCode := '';
GVL_HVCP3.st16CB1HMI.stConfig.sProjectCode := '+EP9-48CB1';
GVL_HVCP3.st16CB1HMI.stConfig.tContactorDelay := T#500MS;
GVL_HVCP3.st16CB1HMI.stConfig.tMotionTimeout := T#50S;
END_METHOD

END_PROGRAM

// ---- POUs/HVCP3/PRG_HVCP3_50CB1.TcPOU
PROGRAM PRG_HVCP3_50CB1
VAR
    // Function Block Instance
    fbDisconnector		: FB_DisconnectorControl;
	
	stDisconnectorIO	: ST_DisconnectorIO;
	
    
    // Başlangıç konfigürasyonu için flag
    bInitDone: BOOL := FALSE;	
END_VAR

IF NOT bInitDone THEN
	bInitDone := TRUE;
	RETURN;
END_IF

//*************************************************************************
// Ana Besleme Ayırıcısı
// +EP6-8CB1
//*************************************************************************
fbDisconnector(
    // Fiziksel Girişler
    bContactorOn_FB 	:= stDisconnectorIO.bContactorOn_FB,
    bContactorOff_FB 	:= stDisconnectorIO.bContactorOff_FB,
    bLimitOn 			:= stDisconnectorIO.bLimitOn,
    bLimitOff 			:= stDisconnectorIO.bLimitOff,
    bThermalFault 		:= stDisconnectorIO.bThermalFault,
    bEarthSwitchOn 		:= stDisconnectorIO.bEarthSwitchOn,
    bEarthSwitchOff 	:= stDisconnectorIO.bEarthSwitchOff,
    bPLCControl 		:= stDisconnectorIO.bPLCControl,
    
    // Güvenlik Girişleri
    bSafetyLoop 		:= GVL_Alarm.bSafetyLoop,
    bInterlock 			:= FALSE,
    
    // Sistem Girişleri
    bMasterReset 		:= GVL_Alarm.bMasterReset,
    
    // HMI Bağlantısı
    stHMI 				:= GVL_HVCP3.st50CB1HMI,
    
    // Fiziksel Çıkışlar
    bContactorOn_Out 	=> stDisconnectorIO.bContactorOn_Out,
    bContactorOff_Out 	=> stDisconnectorIO.bContactorOff_Out
);

METHOD M_Init : BOOL
VAR_INPUT
END_VAR

GVL_HVCP3.st16CB1HMI.stConfig.bEarthSwitchExists := FALSE;
GVL_HVCP3.st16CB1HMI.stConfig.bGrounded := FALSE;
GVL_HVCP3.st16CB1HMI.stConfig.bInterlockEnable := TRUE;
GVL_HVCP3.st16CB1HMI.stConfig.dwOperationLimit := 10000;
GVL_HVCP3.st16CB1HMI.stConfig.nPhaseCount := 3;
GVL_HVCP3.st16CB1HMI.stConfig.rRatedCurrent := 1000.0;
GVL_HVCP3.st16CB1HMI.stConfig.rRatedVoltage := 36000.0;
GVL_HVCP3.st16CB1HMI.stConfig.sProductCode := '';
GVL_HVCP3.st16CB1HMI.stConfig.sProjectCode := '+EP9-12CB1';
GVL_HVCP3.st16CB1HMI.stConfig.tContactorDelay := T#500MS;
GVL_HVCP3.st16CB1HMI.stConfig.tMotionTimeout := T#50S;
END_METHOD

END_PROGRAM

// ---- POUs/HVCP3/PRG_HVCP3_52CB1.TcPOU
PROGRAM PRG_HVCP3_52CB1
VAR
    // Function Block Instance
    fbDisconnector		: FB_DisconnectorControl;
	
	stDisconnectorIO	: ST_DisconnectorIO;
	
    
    // Başlangıç konfigürasyonu için flag
    bInitDone: BOOL := FALSE;	
END_VAR

IF NOT bInitDone THEN
	bInitDone := TRUE;
	RETURN;
END_IF

//*************************************************************************
// Ana Besleme Ayırıcısı
// +EP6-8CB1
//*************************************************************************
fbDisconnector(
    // Fiziksel Girişler
    bContactorOn_FB 	:= stDisconnectorIO.bContactorOn_FB,
    bContactorOff_FB 	:= stDisconnectorIO.bContactorOff_FB,
    bLimitOn 			:= stDisconnectorIO.bLimitOn,
    bLimitOff 			:= stDisconnectorIO.bLimitOff,
    bThermalFault 		:= stDisconnectorIO.bThermalFault,
    bEarthSwitchOn 		:= stDisconnectorIO.bEarthSwitchOn,
    bEarthSwitchOff 	:= stDisconnectorIO.bEarthSwitchOff,
    bPLCControl 		:= stDisconnectorIO.bPLCControl,
    
    // Güvenlik Girişleri
    bSafetyLoop 		:= GVL_Alarm.bSafetyLoop,
    bInterlock 			:= FALSE,
    
    // Sistem Girişleri
    bMasterReset 		:= GVL_Alarm.bMasterReset,
    
    // HMI Bağlantısı
    stHMI 				:= GVL_HVCP3.st52CB1HMI,
    
    // Fiziksel Çıkışlar
    bContactorOn_Out 	=> stDisconnectorIO.bContactorOn_Out,
    bContactorOff_Out 	=> stDisconnectorIO.bContactorOff_Out
);

METHOD M_Init : BOOL
VAR_INPUT
END_VAR

